# B&R Automation Studio project Parker_BMM_ST_V5_3147_V12 (part 24)

#### calib.c
```c
/********************************************************************
 * COPYRIGHT --  B&R China
 ********************************************************************
 * Program: calib
 * File: calib.c
 * Author: lijianjun
 * Created: March 06, 2013
 ********************************************************************
 * Implementation of program calib --- machine calibn control
 ********************************************************************/

#include <bur/plctypes.h>
#include <string.h>

#ifdef _DEFAULT_INCLUDES
#include <AsDefault.h>
#endif

#include "edge.h"               /*edge function                         */
//#include "keyap880.h"
#include "keyap2100.h"
#include "pic_id.h"
/**************************************************************************************
                            Function Declarations
**************************************************************************************/
void CalibCtrl( Mold_typ *pMold);
void CalibRLCtrl( Mold_typ *pMold);

/**************************************************************************************
**     	        		I N I T U P  O F   T H E   T A S K 		 				     **
**************************************************************************************/
_INIT void calib_init ( void )
{
	t_init = 1;         	/* Disable init step: Don't run init step in first cycle */
	t_stop = 1;				/* Enable stop step:  Run stop step in first cycle */

	Init = 0;
}

/**************************************************************************************
        				C Y C L I C   P A R T   O F   T H E   T A S K
**************************************************************************************/

_CYCLIC void calib_cyclic ( void )
{
	if (0 == t_init)                    /*init step: run only one time after resume  init auto course data  */
	{
		t_init = 1;				        /* Disable init step */
		t_stop = 0;

		gTKcalib.Status = 1;

	}/* if(t_init == 0 ) */

	/*auto solution  */
	gTKcalib.Active++;                  /*  task wait status number */
	/*  ---------------------------------- scan code ------------------------------------------ */
	if(1 == gMachineIn.MainControl && gPanelObj.GetPicture != PIC_INIT && gPanelObj.GetPicture != PIC_SCREEN_SAVE )
	{
		/*  key stop or not  */
		gMachineIn.CalibMode = 1;
		if(PIC_OPTION == gPanelObj.GetPicture)
		{
			if(1 == EDGEPOS(gPanelObj.KeyMatric[S$KEYMATRIX_F12],PKeyMatric[S$KEYMATRIX_F12]))
				{
				RMold.AutoStep			   = 30000;
				RMold.ResetStep			= 30000;
				RMold.LowBlow.Step		= 30000;
				RMold.HighBlow.Step		= 30000;
				RMold.BlowPin.Step		= 30000;
				RMold.BlowPin2.Step		= 30000;
				if(RMold.Carriage.Step < 18000 || RMold.Carriage.Step > 19000)RMold.Carriage.Step = 30000;
				RMold.Clamp.Step		   = 30000;
				//	RMold.CoolPin.Step	   = 30000;
				RMold.CoolPinBlow.Step	= 30000;
				RMold.BlowDeflash.Step	= 30000;
				RMold.Cutter.Step		   = 30000;
				RMold.TopDeflash.Step	= 30000;
				RMold.BottomDeflash.Step= 30000;
				RMold.SupportAir.Step	= 30000;
				RMold.SupportSuckAir.Step	= 30000;
				RMold.ExtrLift.Step		= 30000;
				RMold.Lock.Step			= 30000;
				RMold.PullBottom.Step	= 30000;
				RMold.InnerPin.Step	   = 30000;
				RMold.CutNeck.Step	   = 30000;
				//	RMold.Robot.Step	      = 30000;
				RMold.ChuteDeflashBlow.Step = 30000;
				RMold.SubMold.Step	   = 30000;
				RMold.CoolPin2Blow.Step	= 30000;
				RMold.CoolPin3Blow.Step	= 30000;

				gMacOption.Station  = 0;
			}

			if(1 == EDGEPOS(gPanelObj.KeyMatric[S$KEYMATRIX_F13],PKeyMatric[S$KEYMATRIX_F13]))
				{
				LMold.AutoStep			   = 30000;
				LMold.ResetStep			= 30000;
				LMold.LowBlow.Step		= 30000;
				LMold.HighBlow.Step		= 30000;
				LMold.BlowPin.Step		= 30000;
				LMold.BlowPin2.Step		= 30000;
				LMold.CoolPinBlow.Step	= 30000;
				if(LMold.Carriage.Step < 18000 || LMold.Carriage.Step > 19000)LMold.Carriage.Step	= 30000;
				LMold.Clamp.Step		   = 30000;
				//	LMold.CoolPin.Step	   = 30000;
				LMold.BlowDeflash.Step	= 30000;
				LMold.Cutter.Step		   = 30000;
				LMold.TopDeflash.Step	= 30000;
				LMold.BottomDeflash.Step= 30000;
				LMold.SupportAir.Step	= 30000;
				LMold.SupportSuckAir.Step	= 30000;
				LMold.ExtrLift.Step		= 30000;
				LMold.Lock.Step			= 30000;
				LMold.PullBottom.Step	= 30000;
				LMold.InnerPin.Step	   = 30000;
				LMold.CutNeck.Step	   = 30000;
				//	LMold.Robot.Step	      = 30000;
				LMold.ChuteDeflashBlow.Step = 30000;
				LMold.SubMold.Step	   = 30000;
				LMold.CoolPin2Blow.Step	= 30000;
				LMold.CoolPin3Blow.Step	= 30000;

				gMacOption.Station = 1;
			}

			if(1 == EDGEPOS(gPanelObj.KeyMatric[S$KEYMATRIX_F14],PKeyMatric[S$KEYMATRIX_F14]))
				{
				LMold.AutoStep			   = 30000;
				LMold.ResetStep			= 30000;
				LMold.LowBlow.Step		= 30000;
				LMold.HighBlow.Step	   = 30000;
				LMold.BlowPin.Step		= 30000;
				LMold.BlowPin2.Step		= 30000;
				if(LMold.Carriage.Step < 18000 || LMold.Carriage.Step > 19000)LMold.Carriage.Step	= 30000;
				LMold.Clamp.Step		   = 30000;
				//	LMold.CoolPin.Step	   = 30000;
				LMold.CoolPinBlow.Step	= 30000;
				LMold.BlowDeflash.Step	= 30000;
				LMold.Cutter.Step	      = 30000;
				LMold.TopDeflash.Step	= 30000;
				LMold.BottomDeflash.Step= 30000;
				LMold.SupportAir.Step	= 30000;
				LMold.SupportSuckAir.Step	= 30000;
				LMold.ExtrLift.Step		= 30000;
				LMold.Lock.Step			= 30000;
				LMold.PullBottom.Step	= 30000;
				LMold.InnerPin.Step	   = 30000;
				LMold.CutNeck.Step	   = 30000;
				//	LMold.Robot.Step	      = 30000;
				LMold.ChuteDeflashBlow.Step = 30000;
				LMold.SubMold.Step	   = 30000;
				LMold.CoolPin2Blow.Step	= 30000;
				LMold.CoolPin3Blow.Step	= 30000;

				RMold.AutoStep			   = 30000;
				RMold.ResetStep			= 30000;
				RMold.LowBlow.Step		= 30000;
				RMold.HighBlow.Step		= 30000;
				RMold.BlowPin.Step		= 30000;
				RMold.BlowPin2.Step		= 30000;
				if(RMold.Carriage.Step < 18000 || RMold.Carriage.Step > 19000)RMold.Carriage.Step = 30000;
				RMold.Clamp.Step		   = 30000;
				//	RMold.CoolPin.Step  	   = 30000;
				RMold.CoolPinBlow.Step	= 30000;
				RMold.BlowDeflash.Step	= 30000;
				RMold.Cutter.Step		   = 30000;
				RMold.TopDeflash.Step	= 30000;
				RMold.BottomDeflash.Step= 30000;
				RMold.SupportAir.Step	= 30000;
				RMold.SupportSuckAir.Step	= 30000;
				RMold.ExtrLift.Step		= 30000;
				RMold.Lock.Step			= 30000;
				RMold.PullBottom.Step	= 30000;
				RMold.InnerPin.Step	   = 30000;
				RMold.CutNeck.Step   	= 30000;
				//	RMold.Robot.Step	      = 30000;
				RMold.ChuteDeflashBlow.Step = 30000;
				RMold.SubMold.Step	   = 30000;
				RMold.CoolPin2Blow.Step	= 30000;
				RMold.CoolPin3Blow.Step	= 30000;

				gMacOption.Station  = 2;
			}
		}/* if(PIC_OPTION == gPanelObj.GetPicture) */

		if(1 == gMachineFix.Option.bHideLeftStation)
		{
			gMacOption.Station = 1;
			RightOption = 1;
			LeftOption = 0;
		}

		if(1 == LeftOption && 0 == LeftOptionOld)
		{
			RightOption = 0;
			LeftRight   = 0;

			RMold.AutoStep			   = 30000;
			RMold.ResetStep			= 30000;
			RMold.LowBlow.Step		= 30000;
			RMold.HighBlow.Step		= 30000;
			RMold.BlowPin.Step		= 30000;
			RMold.BlowPin2.Step		= 30000;
			if(RMold.Carriage.Step < 18000 || RMold.Carriage.Step > 19000)RMold.Carriage.Step = 30000;
			RMold.Clamp.Step		   = 30000;
			//	RMold.CoolPin.Step	   = 30000;
			RMold.CoolPinBlow.Step	= 30000;
			RMold.BlowDeflash.Step	= 30000;
			RMold.Cutter.Step	   	= 30000;
			RMold.TopDeflash.Step	= 30000;
			RMold.BottomDeflash.Step= 30000;
			RMold.SupportAir.Step	= 30000;
			RMold.SupportSuckAir.Step	= 30000;
			RMold.ExtrLift.Step		= 30000;
			RMold.Lock.Step			= 30000;
			RMold.PullBottom.Step	= 30000;
			RMold.InnerPin.Step	   = 30000;
			RMold.CutNeck.Step	   = 30000;
			//	RMold.Robot.Step	      = 30000;
			RMold.SubMold.Step	   = 30000;
			RMold.ChuteDeflashBlow.Step = 30000;
			RMold.CoolPin2Blow.Step	= 30000;
			RMold.CoolPin3Blow.Step	= 30000;
			gMacOption.Station = 0;
		}

		LeftOptionOld = LeftOption;

		if(1 == RightOption && 0 == RightOptionOld)
		{
			LeftOption  = 0;
			LeftRight   = 0;

			LMold.AutoStep			   = 30000;
			LMold.ResetStep	      = 30000;
			LMold.LowBlow.Step		= 30000;
			LMold.HighBlow.Step		= 30000;
			LMold.BlowPin.Step		= 30000;
			LMold.BlowPin2.Step		= 30000;
			LMold.CoolPinBlow.Step	= 30000;
			if(LMold.Carriage.Step < 18000 || LMold.Carriage.Step > 19000)LMold.Carriage.Step = 30000;
			LMold.Clamp.Step		   = 30000;
			//	LMold.CoolPin.Step	   = 30000;
			LMold.BlowDeflash.Step	= 30000;
			LMold.Cutter.Step		   = 30000;
			LMold.TopDeflash.Step	= 30000;
			LMold.BottomDeflash.Step= 30000;
			LMold.SupportAir.Step	= 30000;
			LMold.SupportSuckAir.Step	= 30000;
			LMold.ExtrLift.Step		= 30000;
			LMold.Lock.Step			= 30000;
			LMold.PullBottom.Step	= 30000;
			LMold.InnerPin.Step	   = 30000;
			LMold.CutNeck.Step	   = 30000;
			//	LMold.Robot.Step	      = 30000;
			LMold.ChuteDeflashBlow.Step = 30000;
			LMold.SubMold.Step	   = 30000;
			LMold.CoolPin2Blow.Step	= 30000;
			LMold.CoolPin3Blow.Step	= 30000;

			gMacOption.Station  = 1;
		}

		RightOptionOld = RightOption;

		if(1 == LeftRight && 0 == LeftRightOld)
		{
			LeftOption  = 0;
			RightOption = 0;

			LMold.AutoStep			   = 30000;
			LMold.ResetStep		   = 30000;
			LMold.LowBlow.Step		= 30000;
			LMold.HighBlow.Step		= 30000;
			LMold.BlowPin.Step		= 30000;
			LMold.BlowPin2.Step		= 30000;
			if(LMold.Carriage.Step < 18000 || LMold.Carriage.Step > 19000)LMold.Carriage.Step = 30000;
			LMold.Clamp.Step		   = 30000;
			//	LMold.CoolPin.Step	   = 30000;
			LMold.CoolPinBlow.Step	= 30000;
			LMold.BlowDeflash.Step	= 30000;
			LMold.Cutter.Step		   = 30000;
			LMold.TopDeflash.Step	= 30000;
			LMold.BottomDeflash.Step= 30000;
			LMold.SupportAir.Step	= 30000;
			LMold.SupportSuckAir.Step	= 30000;
			LMold.ExtrLift.Step		= 30000;
			LMold.Lock.Step			= 30000;
			LMold.PullBottom.Step	= 30000;
			LMold.InnerPin.Step	   = 30000;
			LMold.CutNeck.Step	   = 30000;
			//	LMold.Robot.Step	      = 30000;
			LMold.ChuteDeflashBlow.Step	      = 30000;
			LMold.SubMold.Step	   = 30000;
			LMold.CoolPin2Blow.Step	= 30000;
			LMold.CoolPin3Blow.Step	= 30000;

			RMold.AutoStep			   = 30000;
			RMold.ResetStep			= 30000;
			RMold.LowBlow.Step		= 30000;
			RMold.HighBlow.Step	   = 30000;
			RMold.BlowPin.Step		= 30000;
			RMold.BlowPin2.Step		= 30000;
			if(RMold.Carriage.Step < 18000 || RMold.Carriage.Step > 19000)RMold.Carriage.Step	= 30000;
			RMold.Clamp.Step		   = 30000;
			//	RMold.CoolPin.Step  	   = 30000;
			RMold.CoolPinBlow.Step	= 30000;
			RMold.BlowDeflash.Step	= 30000;
			RMold.Cutter.Step		   = 30000;
			RMold.TopDeflash.Step	= 30000;
			RMold.BottomDeflash.Step= 30000;
			RMold.SupportAir.Step	= 30000;
			RMold.SupportSuckAir.Step	= 30000;
			RMold.ExtrLift.Step		= 30000;
			RMold.Lock.Step			= 30000;
			RMold.PullBottom.Step	= 30000;
			RMold.InnerPin.Step	   = 30000;
			RMold.CutNeck.Step  	   = 30000;
			//	RMold.Robot.Step	      = 30000;
			RMold.ChuteDeflashBlow.Step = 30000;
			RMold.SubMold.Step	   = 30000;
			RMold.CoolPin2Blow.Step	= 30000;
			RMold.CoolPin3Blow.Step	= 30000;

			gMacOption.Station = 2;
		}

		LeftRightOld = LeftRight;

		if(0 == gMacOption.Station)
		{
			LeftOption = 1;
			RightOption = 0;
			LeftRight = 0;
		}

		if(1 == gMacOption.Station)
		{
			LeftOption  = 0;
			RightOption = 1;
			LeftRight   = 0;
		}

		if(2 == gMacOption.Station)
		{
			LeftOption  = 0;
			RightOption = 0;
			LeftRight   = 1;
		}

		if(1 == gMachineIn.CalibMode && 0 == gMachineIn.SafeCalibPressure)
		{
			/* ---------------- 左右模动作 ---------------- */
			//1 = 正常模式    0 = hold to run
			if((0 == RightOption) && (1 == LeftOption))
			{
				CalibCtrl(&LMold);
			}

			if((1 == RightOption) && (0 == LeftOption))
			{
				CalibCtrl(&RMold);
			}

			if ((0 == RightOption) && (0 == LeftOption))
			{
				CalibRLCtrl(&RMold);
			}

		}/* if(1 == gMachineIn.CalibMode) */
	}/* if(1 == gMachineIn.MainControl && gPanelObj.GetPicture != PIC_INIT && gPanelObj.GetPicture != PIC_SCREEN_SAVE) */
	/*  --------------------------------------------------------------------------------------- */

	if (1 == gTKcalib.Stop)   /* enable stop step */
	{
		t_stop        = 1;
		gTKcalib.Stop = 0;
	}

	/* auto solution end */
	if(1 == t_stop)
	{
		//	memset(&LMold.ValveOut,0,sizeof(LMold.ValveOut));
		//	memset(&RMold.ValveOut,0,sizeof(RMold.ValveOut));

		//		memset(&gMachineOut.LMold,0,sizeof(gMachineOut.LMold));
		//    	memset(&gMachineOut.RMold,0,sizeof(gMachineOut.RMold));

//		memset(&LMold.ValveOut.ClampCls,0,sizeof(LMold.ValveOut)-12);
//		memset(&RMold.ValveOut.ClampCls,0,sizeof(RMold.ValveOut)-12);

		LMold.BottomDeflash.Step = 30000;
		RMold.BottomDeflash.Step = 30000;

		LMold.HighBlow.Step = 30000;
		RMold.HighBlow.Step = 30000;

		LMold.LowBlow.Step = 30000;
		RMold.LowBlow.Step = 30000;

		LMold.BlowPin.Step = 30000;
		RMold.BlowPin.Step = 30000;

		LMold.BlowPin2.Step = 30000;
		RMold.BlowPin2.Step = 30000;

		LMold.Clamp.Step = 30000;
		RMold.Clamp.Step = 30000;

		LMold.Carriage.Step = 30000;
		RMold.Carriage.Step = 30000;

		LMold.TopDeflash.Step = 30000;
		RMold.TopDeflash.Step = 30000;

		LMold.Plate.Step = 30000;/*Albert*/
		RMold.Plate.Step = 30000;/*Albert*/

		LMold.Carriage.v_set = 0;
		RMold.Carriage.v_set = 0;

		LMold.Clamp.v_set = 0;
		RMold.Clamp.v_set = 0;

		LMold.Clamp.p_set = 0;/*Albert*/
		RMold.Clamp.p_set = 0;/*Albert*/

		LMold.BlowPin.v_set = 0;
		RMold.BlowPin.v_set = 0;

		LMold.TopDeflash.p_set = 0;/*Albert*/
		RMold.TopDeflash.p_set = 0;/*Albert*/

		LMold.Plate.p_set = 0;/*Albert*/
		RMold.Plate.p_set = 0;/*Albert*/

		LMold.BottomDeflash.p_set =0;
		RMold.BottomDeflash.p_set =0;

		LMold.SubMold.Step =30000;
		RMold.SubMold.Step =30000;

		LMold.BottomSubMold.Step =30000;
		RMold.BottomSubMold.Step =30000;

		LMold.SubMold.p_set =0;
		RMold.SubMold.p_set =0;

		LMold.BottomSubMold.p_set =0;
		RMold.BottomSubMold.p_set =0;

		LMold.RobotOpnCls.Step = 30000;
		RMold.RobotOpnCls.Step = 30000;

		LMold.Robot.Step = 30000;
		RMold.Robot.Step = 30000;

		t_init         = 0;                 /* next resume ,enable init step */
		gTKcalib.Status = 0;
		ST_tmp_suspend(0);
	} /* if (t_stop==1) */

}

/* ------------------------------------------------------------------*/
void CalibCtrl( Mold_typ *pMold)
{
	if (1==gMacOption.Station) /*Right mold*/
	{
		/* -------------------  Carriage up   ----------------------*/
		if(1 == EDGEPOS(gPanelObj.KeyMatric[S$KEYMATRIX_CARRIAGE_UP ],PKeyMatric[S$KEYMATRIX_CARRIAGE_UP ]))
		{
			if(1 == gMachineOut.OilPump)
			{
				if( 1 == pMold->TransDIn.ClampOpnLimit || (1 == pMold->TransDIn.BlowPinUpLimit && 1 == pMold->TransDIn.BlowPin2UpLimit))
				{
					if(	1 == pMold->TransDIn.TopDeflashBwLimit
						&& 1 == pMold->TransDIn.BottomDeflashBwLimit
						&& 1 == pMold->TransDIn.SubMoldClsLimit && 1 == pMold->TransDIn.BottomSubMoldClsLimit
						&& 1 == pMold->TransDIn.HookPinBwLimit)
					{
						if(((pMold == & LMold) && 1 == RMold.TransDIn.CarriageBwLimit)
							||((pMold == & RMold) && (1 == gMachineFix.Option.bHideLeftStation || 1 == LMold.TransDIn.CarriageBwLimit)))
						{
							pMold->Carriage.Step = 5000;       /* Carriage up calibration */
						}
						else
						{
							if(pMold == & LMold)
							{
								gImply.RCarriageBw = !RMold.TransDIn.CarriageBwLimit;
							}
							else
							{
								gImply.LCarriageBw = !LMold.TransDIn.CarriageBwLimit;
							}
						}
					}
					else
					{
						if(pMold == & LMold)
						{
							gImply.LTopDeflashBw 	= !pMold->TransDIn.TopDeflashBwLimit;
							gImply.LBottomDeflashBw = !pMold->TransDIn.BottomDeflashBwLimit;
							gImply.LSubMoldFw 		= !pMold->TransDIn.SubMoldClsLimit;
							gImply.LBottomSubMoldFw	= !pMold->TransDIn.BottomSubMoldClsLimit;
							gImply.LHookPinBw 		= !pMold->TransDIn.HookPinBwLimit;

						}
						else
						{
							gImply.RTopDeflashBw 	= !pMold->TransDIn.TopDeflashBwLimit;
							gImply.RBottomDeflashBw = !pMold->TransDIn.BottomDeflashBwLimit;
							gImply.RSubMoldFw 		= !pMold->TransDIn.SubMoldClsLimit;
							gImply.RBottomSubMoldFw	= !pMold->TransDIn.BottomSubMoldClsLimit;
							gImply.RHookPinBw 		= !pMold->TransDIn.HookPinBwLimit;
						}
					}
				}
				else
				{
					if(pMold == & LMold)
					{
						gImply.LClampOpn     = !pMold->TransDIn.ClampOpnLimit;
						gImply.LPinUp    	 = !pMold->TransDIn.BlowPinUpLimit;
						gImply.LPin2Up    	 = !pMold->TransDIn.BlowPin2UpLimit;
					}
					else
					{
						gImply.RClampOpn     = !pMold->TransDIn.ClampOpnLimit;
						gImply.RPinUp    	 = !pMold->TransDIn.BlowPinUpLimit;
						gImply.RPin2Up    	 = !pMold->TransDIn.BlowPin2UpLimit;
					}

				}
			}
			else
			{
				gImply.OilPumpNotOn  = !gMachineOut.OilPump;
			}
		}/* if(1 == EDGEPOS(gPanelObj.KeyMatric[S$KEYMATRIX_CARRIAGE_UP  ],PKeyMatric[S$KEYMATRIX_CARRIAGE_UP  ])) */

		if(1 == EDGENEG(gPanelObj.KeyMatric[S$KEYMATRIX_CARRIAGE_UP ],NKeyMatric[S$KEYMATRIX_CARRIAGE_UP]))
		{
			pMold->Carriage.Step = 20000;
		}

		/* -------------------  Carriage down   ----------------------*/
		if(1 == EDGEPOS(gPanelObj.KeyMatric[S$KEYMATRIX_CARRIAGE_DN ],PKeyMatric[S$KEYMATRIX_CARRIAGE_DN ]))
		{
			if(1 == gMachineOut.OilPump)
			{
				if(1 == pMold->TransDIn.BlowPinUpLimit && 1 == pMold->TransDIn.BlowPin2UpLimit)
				{
					if( 1 == pMold->TransDIn.TopDeflashBwLimit
						&& 1 == pMold->TransDIn.BottomDeflashBwLimit
						&& 1 == pMold->TransDIn.CoolPinUpLimit && 1 == pMold->TransDIn.CoolPin2UpLimit && 1==pMold->TransDIn.CoolPin3UpLimit
						&& 1 == pMold->TransDIn.RobotBwLimit
						&& 1 == pMold->TransDIn.ExtRobotUpLmit
						&& 1 == pMold->TransDIn.HookPinBwLimit)
					{
						pMold->Carriage.Step = 15000;       /* Carriage down calibration */
					}
					else
					{
						if(pMold == & LMold)
						{
							gImply.LTopDeflashBw = ! pMold->TransDIn.TopDeflashBwLimit;
							gImply.LBottomDeflashBw = ! pMold->TransDIn.BottomDeflashBwLimit;
							gImply.LCoolPinUp	= !pMold->TransDIn.CoolPinUpLimit;
							gImply.LCoolPin2Up	= !pMold->TransDIn.CoolPin2UpLimit;
							gImply.LCoolPin3Up	= !pMold->TransDIn.CoolPin3UpLimit;
							gImply.LRobotBw		= !pMold->TransDIn.RobotBwLimit;

							gImply.LExtRobotUp 		= !pMold->TransDIn.ExtRobotUpLmit;
							gImply.LHookPinBw 		= !pMold->TransDIn.HookPinBwLimit;
						}
						else
						{
							gImply.RTopDeflashBw = !pMold->TransDIn.TopDeflashBwLimit;
							gImply.RBottomDeflashBw = ! pMold->TransDIn.BottomDeflashBwLimit;
							gImply.RCoolPinUp	= !pMold->TransDIn.CoolPinUpLimit;
							gImply.RCoolPin2Up	= !pMold->TransDIn.CoolPin2UpLimit;
							gImply.RCoolPin3Up	= !pMold->TransDIn.CoolPin3UpLimit;
							gImply.RRobotBw		= !pMold->TransDIn.RobotBwLimit;

							gImply.RExtRobotUp 		= !pMold->TransDIn.ExtRobotUpLmit;
							gImply.RHookPinBw 		= !pMold->TransDIn.HookPinBwLimit;
						}

					}
				}
				else
				{
					if(pMold == & LMold)
					{
						gImply.LPinUp        = !pMold->TransDIn.BlowPinUpLimit;
						gImply.LPin2Up       = !pMold->TransDIn.BlowPin2UpLimit;
					}
					else
					{
						gImply.RPinUp        = !pMold->TransDIn.BlowPinUpLimit;
						gImply.RPin2Up       = !pMold->TransDIn.BlowPin2UpLimit;
					}

				}
			}
			else
			{
				gImply.OilPumpNotOn  = !gMachineOut.OilPump;
			}

		}/* if(1 == EDGEPOS(gPanelObj.KeyMatric[S$KEYMATRIX_CARRIAGE_DN ],PKeyMatric[S$KEYMATRIX_CARRIAGE_DN ]))*/

		if(1 == EDGENEG(gPanelObj.KeyMatric[S$KEYMATRIX_CARRIAGE_DN ],NKeyMatric[S$KEYMATRIX_CARRIAGE_DN ]))
		{
			pMold->Carriage.Step = 20000;
		}
	}
	/*-------------------------------------------------------------------------------------------------------------------*/
	if (0==gMacOption.Station) /*left mold*/
	{
		/* -------------------  Carriage up   ----------------------*/
		if(1 == EDGEPOS(gPanelObj.KeyMatric[S$KEYMATRIX_CARRIAGE_DN ],PKeyMatric[S$KEYMATRIX_CARRIAGE_DN ]))
		{
			if(1 == gMachineOut.OilPump)
			{
				if( 1 == pMold->TransDIn.ClampOpnLimit || (1 == pMold->TransDIn.BlowPinUpLimit && 1 == pMold->TransDIn.BlowPin2UpLimit))
				{
					if(	1 == pMold->TransDIn.TopDeflashBwLimit
						&& 1 == pMold->TransDIn.BottomDeflashBwLimit
						&& 1 == pMold->TransDIn.SubMoldClsLimit && 1 == pMold->TransDIn.BottomSubMoldClsLimit
						&& 1 == pMold->TransDIn.HookPinBwLimit)
					{
						if(((pMold == & LMold) && 1 == RMold.TransDIn.CarriageBwLimit)
							||((pMold == & RMold) && (1 == gMachineFix.Option.bHideLeftStation || 1 == LMold.TransDIn.CarriageBwLimit)))
						{
							pMold->Carriage.Step = 5000;       /* Carriage up calibration */
						}
						else
						{
							if(pMold == & LMold)
							{
								gImply.RCarriageBw = !RMold.TransDIn.CarriageBwLimit;
							}
							else
							{
								gImply.LCarriageBw = !LMold.TransDIn.CarriageBwLimit;
							}
						}
					}
					else
					{
						if(pMold == & LMold)
						{
							gImply.LTopDeflashBw 	= ! pMold->TransDIn.TopDeflashBwLimit;
							gImply.LBottomDeflashBw = !pMold->TransDIn.BottomDeflashBwLimit;
							gImply.LSubMoldFw 		= !pMold->TransDIn.SubMoldClsLimit;
							gImply.LBottomSubMoldFw	= !pMold->TransDIn.BottomSubMoldClsLimit;
							gImply.LHookPinBw 		= !pMold->TransDIn.HookPinBwLimit;
						}
						else
						{
							gImply.RTopDeflashBw 	= ! pMold->TransDIn.TopDeflashBwLimit;
							gImply.RBottomDeflashBw = !pMold->TransDIn.BottomDeflashBwLimit;
							gImply.RSubMoldFw 		= !pMold->TransDIn.SubMoldClsLimit;
							gImply.RBottomSubMoldFw	= !pMold->TransDIn.BottomSubMoldClsLimit;
							gImply.RHookPinBw 		= !pMold->TransDIn.HookPinBwLimit;
						}

					}
				}
				else
				{
					if(pMold == & LMold)
					{
						gImply.LClampOpn     = !pMold->TransDIn.ClampOpnLimit;
						gImply.LPinUp    	 = !pMold->TransDIn.BlowPinUpLimit;
						gImply.LPin2Up    	 = !pMold->TransDIn.BlowPin2UpLimit;
					}
					else
					{
						gImply.RClampOpn     = !pMold->TransDIn.ClampOpnLimit;
						gImply.RPinUp    	 = !pMold->TransDIn.BlowPinUpLimit;
						gImply.RPin2Up    	 = !pMold->TransDIn.BlowPin2UpLimit;
					}

				}
			}
			else
			{
				gImply.OilPumpNotOn  = !gMachineOut.OilPump;
			}
		}/* if(1 == EDGEPOS(gPanelObj.KeyMatric[S$KEYMATRIX_CARRIAGE_DN  ],PKeyMatric[S$KEYMATRIX_CARRIAGE_DN  ])) */

		if(1 == EDGENEG(gPanelObj.KeyMatric[S$KEYMATRIX_CARRIAGE_DN ],NKeyMatric[S$KEYMATRIX_CARRIAGE_DN]))
		{
			pMold->Carriage.Step = 20000;
		}

		/* -------------------  Carriage down   ----------------------*/
		if(1 == EDGEPOS(gPanelObj.KeyMatric[S$KEYMATRIX_CARRIAGE_UP],PKeyMatric[S$KEYMATRIX_CARRIAGE_UP ]))
		{
			if(1 == gMachineOut.OilPump)
			{
				if(1 == pMold->TransDIn.BlowPinUpLimit && 1 == pMold->TransDIn.BlowPin2UpLimit)
				{
					if( 1 == pMold->TransDIn.TopDeflashBwLimit
						&& 1 == pMold->TransDIn.BottomDeflashBwLimit
						&& 1 == pMold->TransDIn.CoolPinUpLimit && 1 == pMold->TransDIn.CoolPin2UpLimit && 1==pMold->TransDIn.CoolPin3UpLimit
						&& 1 == pMold->TransDIn.ExtRobotUpLmit
						&& 1 == pMold->TransDIn.HookPinBwLimit)
					{
						pMold->Carriage.Step = 15000;       /* Carriage down calibration */
					}
					else
					{
						if(pMold == & LMold)
						{
							gImply.LPinUp        = !pMold->TransDIn.BlowPinUpLimit;
							gImply.LTopDeflashBw = ! pMold->TransDIn.TopDeflashBwLimit;
							gImply.LBottomDeflashBw = ! pMold->TransDIn.BottomDeflashBwLimit;
							gImply.LCoolPinUp	= !pMold->TransDIn.CoolPinUpLimit;
							gImply.LCoolPin2Up	= !pMold->TransDIn.CoolPin2UpLimit;
							gImply.LCoolPin3Up	= !pMold->TransDIn.CoolPin3UpLimit;

							gImply.LExtRobotUp 		= !pMold->TransDIn.ExtRobotUpLmit;
							gImply.LHookPinBw 		= !pMold->TransDIn.HookPinBwLimit;

						}
						else
						{
							gImply.RPinUp        = !pMold->TransDIn.BlowPinUpLimit;
							gImply.RTopDeflashBw = !pMold->TransDIn.TopDeflashBwLimit;
							gImply.RBottomDeflashBw = ! pMold->TransDIn.BottomDeflashBwLimit;
							gImply.RCoolPinUp	= !pMold->TransDIn.CoolPinUpLimit;
							gImply.RCoolPin2Up	= !pMold->TransDIn.CoolPin2UpLimit;
							gImply.RCoolPin3Up	= !pMold->TransDIn.CoolPin3UpLimit;

							gImply.RExtRobotUp 		= !pMold->TransDIn.ExtRobotUpLmit;
							gImply.RHookPinBw 		= !pMold->TransDIn.HookPinBwLimit;

						}

					}
				}
				else
				{
					if(pMold == & LMold)
					{
						gImply.LPinUp        = !pMold->TransDIn.BlowPinUpLimit;
						gImply.LPin2Up       = !pMold->TransDIn.BlowPin2UpLimit;
					}
					else
					{
						gImply.RPinUp        = !pMold->TransDIn.BlowPinUpLimit;
						gImply.RPin2Up       = !pMold->TransDIn.BlowPin2UpLimit;
					}

				}
			}
			else
			{
				gImply.OilPumpNotOn  = !gMachineOut.OilPump;
			}

		}/* if(1 == EDGEPOS(gPanelObj.KeyMatric[S$KEYMATRIX_CARRIAGE_UP ],PKeyMatric[S$KEYMATRIX_CARRIAGE_UP ]))*/

		if(1 == EDGENEG(gPanelObj.KeyMatric[S$KEYMATRIX_CARRIAGE_UP ],NKeyMatric[S$KEYMATRIX_CARRIAGE_UP ]))
		{
			pMold->Carriage.Step = 20000;
		}
	}

	/*-------------------------------------------------------------------------------------------------------------------*/

	/* -------------------  open  clamp  ----------------------*/
	if(1 == EDGEPOS(gPanelObj.KeyMatric[S$KEYMATRIX_CLAMP_OPN ],PKeyMatric[S$KEYMATRIX_CLAMP_OPN ]))
	{
		if(1 == gMachineOut.OilPump)
		{
			if( 1 == pMold->TransDIn.TopDeflashBwLimit
				&& 1 == pMold->TransDIn.BottomDeflashBwLimit
				&& 1 == pMold->TransDIn.ExtRobotUpLmit)
			{
				pMold->Clamp.Step = 15000;		/*   clamp open calibration   */
			}
			else
			{
				if(pMold == & LMold)
				{
					gImply.LTopDeflashBw 	= !pMold->TransDIn.TopDeflashBwLimit;
					gImply.LBottomDeflashBw = !pMold->TransDIn.BottomDeflashBwLimit;

					gImply.LExtRobotUp 		= !pMold->TransDIn.ExtRobotUpLmit;
				}
				else
				{
					gImply.RTopDeflashBw 	= ! pMold->TransDIn.TopDeflashBwLimit;
					gImply.RBottomDeflashBw = ! pMold->TransDIn.BottomDeflashBwLimit;

					gImply.RExtRobotUp 		= !pMold->TransDIn.ExtRobotUpLmit;

				}
			}
		}
		else
		{
			gImply.OilPumpNotOn  = !gMachineOut.OilPump;
		}

	}

	if(1 == EDGENEG(gPanelObj.KeyMatric[S$KEYMATRIX_CLAMP_OPN ],NKeyMatric[S$KEYMATRIX_CLAMP_OPN ]))
	{
		if(pMold == & LMold)
		{
			gLClampOpnFlag_Calib =0;
		}
		else
		{
			gRClampOpnFlag_Calib =0;
		}

		pMold->Clamp.Step = 20000;
	}

	/* -------------------  close  clamp  ----------------------*/
	if(1 == EDGEPOS(gPanelObj.KeyMatric[S$KEYMATRIX_CLAMP_CLS ],PKeyMatric[S$KEYMATRIX_CLAMP_CLS ]))
	{
		if(1 == gMachineOut.OilPump)
		{
			if(1 == pMold->TransDIn.CarriageFwLimit || (1 == pMold->TransDIn.BlowPinUpLimit && 1 == pMold->TransDIn.BlowPin2UpLimit))
			{
				if( 1 == pMold->TransDIn.CoolPinUpLimit
					&& 1 == pMold->TransDIn.SubMoldClsLimit
					&& 1 == pMold->TransDIn.BottomSubMoldClsLimit
					&& 1 == pMold->TransDIn.RobotBwLimit)
				{
					pMold->Clamp.Step = 5000;		/*   clamp close calibration   */
				}
				else
				{
					if(pMold == & LMold)
					{
						gImply.LCoolPinUp = !pMold->TransDIn.CoolPinUpLimit;

						gImply.LSubMoldFw 		= !pMold->TransDIn.SubMoldClsLimit;
						gImply.LBottomSubMoldFw	= !pMold->TransDIn.BottomSubMoldClsLimit;
						gImply.LRobotBw		= !pMold->TransDIn.RobotBwLimit;

					}
					else
					{
						gImply.RCoolPinUp = !pMold->TransDIn.CoolPinUpLimit;

						gImply.RSubMoldFw 		= !pMold->TransDIn.SubMoldClsLimit;
						gImply.RBottomSubMoldFw = !pMold->TransDIn.BottomSubMoldClsLimit;
						gImply.RRobotBw		= !pMold->TransDIn.RobotBwLimit;

					}/* if(pMold == & LMold) */
				}
			}
			else
			{
				if(pMold == & LMold)
				{
					gImply.LCarriageFw	 = !pMold->TransDIn.CarriageFwLimit;
					gImply.LPinUp        = !pMold->TransDIn.BlowPinUpLimit;
					gImply.LPin2Up       = !pMold->TransDIn.BlowPin2UpLimit;
				}
				else
				{
					gImply.RCarriageFw	 = !pMold->TransDIn.CarriageFwLimit;
					gImply.RPinUp        = !pMold->TransDIn.BlowPinUpLimit;
					gImply.RPin2Up       = !pMold->TransDIn.BlowPin2UpLimit;
				}
			}
		}
		else
		{
			gImply.OilPumpNotOn  = !gMachineOut.OilPump;
		}
	}

	if(1 == EDGENEG(gPanelObj.KeyMatric[S$KEYMATRIX_CLAMP_CLS ],NKeyMatric[S$KEYMATRIX_CLAMP_CLS ]))
		{
		if(pMold == & LMold)
		{
			gLClampOpnFlag_Calib =0;
		}
		else
		{
			gRClampOpnFlag_Calib =0;
		}
		pMold->Clamp.Step = 20000;
	}

	/* -------------------   blow pin up  ----------------------*/
	if(1 == EDGEPOS(gPanelObj.KeyMatric[S$KEYMATRIX_BLOWPIN_UP ],PKeyMatric[S$KEYMATRIX_BLOWPIN_UP ]))
	{
		if (1 == gMachineOut.OilPump)
		{
			if(pMold->Option.BlowPin)
			{
				pMold->BlowPin.Step = 15000;
			}

			if(pMold->Option.BlowPin2)
			{
				pMold->BlowPin2.Step = 15000;
			}
		}
		else
		{
			gImply.OilPumpNotOn  = !gMachineOut.OilPump;
		}
	}

	if(1 == EDGENEG(gPanelObj.KeyMatric[S$KEYMATRIX_BLOWPIN_UP ],NKeyMatric[S$KEYMATRIX_BLOWPIN_UP ]))
	{
		pMold->BlowPin.Step = 20000;
		pMold->BlowPin2.Step = 20000;
	}
	/* -------------------   blow pin down  ----------------------*/
	if(1 == EDGEPOS(gPanelObj.KeyMatric[S$KEYMATRIX_BLOWPIN_DN ],PKeyMatric[S$KEYMATRIX_BLOWPIN_DN ]))
	{
		if(1 == gMachineOut.OilPump)
		{
			if(( 1 == pMold->TransDIn.CarriageFwLimit || 1 == pMold->TransDIn.CarriageBwLimit) )
			{
				if(1 == pMold->TransDIn.SubMoldClsLimit
					&& 1 == pMold->TransDIn.BottomSubMoldClsLimit )
				{
					if(pMold->Option.BlowPin)
					{
						pMold->BlowPin.Step = 5000;	/*  blow pin down  */
					}

					if(pMold->Option.BlowPin2)
					{
						pMold->BlowPin2.Step = 5000; /*  blow pin down  */
					}
				}
				else
				{
					if(pMold == & LMold)
					{
						gImply.LSubMoldFw 		= !pMold->TransDIn.SubMoldClsLimit;
						gImply.LBottomSubMoldFw = !pMold->TransDIn.BottomSubMoldClsLimit;

					}
					else
					{
						gImply.RSubMoldFw 		= !pMold->TransDIn.SubMoldClsLimit;
						gImply.RBottomSubMoldFw = !pMold->TransDIn.BottomSubMoldClsLimit;

					}
				}
			}
			else
			{
				if(pMold == & LMold)
				{
					gImply.LCarriageFwBw = !(pMold->TransDIn.CarriageBwLimit || pMold->TransDIn.CarriageFwLimit);
				}
				else
				{
					gImply.RCarriageFwBw = !(pMold->TransDIn.CarriageBwLimit || pMold->TransDIn.CarriageFwLimit);
				}
			}
		}
		else
		{
			gImply.OilPumpNotOn  = !gMachineOut.OilPump;
		}
	}
	if(1 == EDGENEG(gPanelObj.KeyMatric[S$KEYMATRIX_BLOWPIN_DN   ],NKeyMatric[S$KEYMATRIX_BLOWPIN_DN ]))
	{
		pMold->BlowPin.Step = 20000;
		pMold->BlowPin2.Step = 20000;
	}

	/* ------------------------------  pin part forward ----------------------------- */
	if(1 == EDGEPOS(gPanelObj.KeyMatric[S$KEYMATRIX_PIN_PART_FW ],PKeyMatric[S$KEYMATRIX_PIN_PART_FW ]))
		{
		if(pMold->Option.PinPart)
		{
			if(1 == pMold->TransDIn.BlowPinUpLimit)
			{
				pMold->PinPart.Step = 300;
			}
			else
			{
				if(pMold == & LMold)
				{
					gImply.LPinUp = !pMold->TransDIn.BlowPinUpLimit;
				}
				else
				{
					gImply.RPinUp = !pMold->TransDIn.BlowPinUpLimit;
				}
			}
		}
	}

	if(1 == EDGENEG(gPanelObj.KeyMatric[S$KEYMATRIX_PIN_PART_FW ],NKeyMatric[S$KEYMATRIX_PIN_PART_FW ]))
		{
		pMold->PinPart.Step = 20000;
	}

	/* ------------------------------  pin part backward ----------------------------- */
	if(1 == EDGEPOS(gPanelObj.KeyMatric[S$KEYMATRIX_PIN_PART_BW   ],PKeyMatric[S$KEYMATRIX_PIN_PART_BW   ]))
	{
		if(pMold->Option.PinPart)
		{
			if(1 == pMold->TransDIn.BlowPinUpLimit)
			{
				pMold->PinPart.Step = 10300;
			}
			else
			{
				if(pMold == & LMold)
				{
					gImply.LPinUp = !pMold->TransDIn.BlowPinUpLimit;
				}
				else
				{
					gImply.RPinUp = !pMold->TransDIn.BlowPinUpLimit;
				}
			}
		}
	}

	if(1 == EDGENEG(gPanelObj.KeyMatric[S$KEYMATRIX_PIN_PART_BW   ],NKeyMatric[S$KEYMATRIX_PIN_PART_BW   ]))
	{
		pMold->PinPart.Step = 20000;
	}

	/* ------------------------------  Sub mold open ----------------------------- */
	if(1 == EDGEPOS(gPanelObj.KeyMatric[S$KEYMATRIX_SUBMOLD_OPN   ],PKeyMatric[S$KEYMATRIX_SUBMOLD_OPN   ]))
	{
		if(1 == pMold->Option.SubMold )
		{
			if(1 == gMachineOut.OilPump)
			{
				if (1==pMold->Clamp.OpnOverHalf && 1 == pMold->TransDIn.CarriageBwLimit) // 大於微開模
				{
					pMold->SubMold.Step = 15000;
				}
				else
				{
					if(pMold == & LMold)
					{
						gImply.L_SubmoldOut_Clamp = !pMold->Clamp.OpnOverHalf;
						gImply.LCarriageBw = !pMold->TransDIn.CarriageBwLimit;
					}
					else
					{
						gImply.R_SubmoldOut_Clamp = !pMold->Clamp.OpnOverHalf;
						gImply.RCarriageBw = !pMold->TransDIn.CarriageBwLimit;
					}
				}

			}
			else
			{
				gImply.OilPumpNotOn  = !gMachineOut.OilPump;
			}
		}
		else
		{
			gImply.NoFunction = 1;
		}
	}

	if(1 == EDGENEG(gPanelObj.KeyMatric[S$KEYMATRIX_SUBMOLD_OPN   ],NKeyMatric[S$KEYMATRIX_SUBMOLD_OPN   ]))
	{
		pMold->SubMold.Step = 20000;
	}

	/* ------------------------------  sub mold close ----------------------------- */
	if(1 == EDGEPOS(gPanelObj.KeyMatric[S$KEYMATRIX_SUBMOLD_CLS   ],PKeyMatric[S$KEYMATRIX_SUBMOLD_CLS   ]))
	{
		if(pMold->Option.SubMold)
		{
			if(1 == gMachineOut.OilPump)
			{
				pMold->SubMold.Step = 5000;
			}
			else
			{
				gImply.OilPumpNotOn  = !gMachineOut.OilPump;
			}
		}
		else
		{
			gImply.NoFunction = 1;
		}
	}

	if(1 == EDGENEG(gPanelObj.KeyMatric[S$KEYMATRIX_SUBMOLD_CLS   ],NKeyMatric[S$KEYMATRIX_SUBMOLD_CLS   ]))
	{
		pMold->SubMold.Step = 20000;
	}

	/* ------------------------------  Bottom Sub mold open ----------------------------- */
	if(1 == EDGEPOS(gPanelObj.KeyMatric[S$KEYMATRIX_BOTSUBMOLD_OPN  ],PKeyMatric[S$KEYMATRIX_BOTSUBMOLD_OPN  ]))
	{
		if(pMold->Option.BottomSubMold)
		{
			if(1 == gMachineOut.OilPump)
			{
				if (1 == pMold->Clamp.OpnOverHalf && 1 == pMold->TransDIn.CarriageBwLimit)
				{
					pMold->BottomSubMold.Step = 15000;
				}
				else
				{
					if(pMold == & LMold)
					{
						gImply.L_SubmoldOut_Clamp = !pMold->Clamp.OpnOverHalf;
						gImply.LCarriageBw = !pMold->TransDIn.CarriageBwLimit;
					}
					else
					{
						gImply.R_SubmoldOut_Clamp = !pMold->Clamp.OpnOverHalf;
						gImply.RCarriageBw = !pMold->TransDIn.CarriageBwLimit;
					}
				}
			}
			else
			{
				gImply.OilPumpNotOn  = !gMachineOut.OilPump;
			}
		}
		else
		{
			gImply.NoFunction = 1;
		}
	}

	if(1 == EDGENEG(gPanelObj.KeyMatric[S$KEYMATRIX_BOTSUBMOLD_OPN  ],NKeyMatric[S$KEYMATRIX_BOTSUBMOLD_OPN  ]))
	{
		pMold->BottomSubMold.Step = 20000;
	}

	/* ------------------------------ Bottom sub mold close ----------------------------- */
	if(1 == EDGEPOS(gPanelObj.KeyMatric[S$KEYMATRIX_BOTSUBMOLD_CLS  ],PKeyMatric[S$KEYMATRIX_BOTSUBMOLD_CLS  ]))
	{
		if(pMold->Option.BottomSubMold)
		{
			if(1 == gMachineOut.OilPump)
			{
				pMold->BottomSubMold.Step = 5000;
			}
			else
			{
				gImply.OilPumpNotOn  = !gMachineOut.OilPump;
			}
		}
		else
		{
			gImply.NoFunction = 1;
		}
	}
	if(1 == EDGENEG(gPanelObj.KeyMatric[S$KEYMATRIX_BOTSUBMOLD_CLS  ],NKeyMatric[S$KEYMATRIX_BOTSUBMOLD_CLS  ]))
	{
		pMold->BottomSubMold.Step = 20000;
	}

	/* ------------------------------  Screw forward ----------------------------- */
	if(1 == EDGEPOS(gPanelObj.KeyMatric[S$KEYMATRIX_SCREW_FW   ],PKeyMatric[S$KEYMATRIX_SCREW_FW   ]))
	{
		pMold->Screw.Step = 300;
	}

	if(1 == EDGENEG(gPanelObj.KeyMatric[S$KEYMATRIX_SCREW_FW   ],NKeyMatric[S$KEYMATRIX_SCREW_FW   ]))
	{
		pMold->Screw.Step = 20000;
	}

	/* ------------------------------  screw backward ----------------------------- */
	if(1 == EDGEPOS(gPanelObj.KeyMatric[S$KEYMATRIX_SCREW_BW   ],PKeyMatric[S$KEYMATRIX_SCREW_BW   ]))
	{
		pMold->Screw.Step = 10300;
	}

	if(1 == EDGENEG(gPanelObj.KeyMatric[S$KEYMATRIX_SCREW_BW   ],NKeyMatric[S$KEYMATRIX_SCREW_BW   ]))
	{
		pMold->Screw.Step = 20000;
	}

	/* ------------------------------  Top Deflasher forward ----------------------------- */
	if(1 == EDGEPOS(gPanelObj.KeyMatric[S$KEYMATRIX_TOP_DEFLASH_FW  ],PKeyMatric[S$KEYMATRIX_TOP_DEFLASH_FW  ]))
	{
		if(pMold->Option.TopDeflash)
		{
			if(1 == gMachineOut.OilPump)
			{
				if(1 == pMold->TransDIn.CarriageBwLimit
					&& 1 == pMold->Clamp.ClsPos
					&& 1 == pMold->TransDIn.TopDeflashOpnLimit
					&& 1 == pMold->TransDIn.CoolPinUpLimit)
				{
					pMold->TopDeflash.Step = 5000;
				}
				else
				{
					if(pMold == & LMold)
					{
						gImply.LCarriageBw	= !pMold->TransDIn.CarriageBwLimit;
						gImply.LClampCls	= !pMold->Clamp.ClsPos;
						gImply.LTopDeflashOpn	= !pMold->TransDIn.TopDeflashOpnLimit;
						gImply.LCoolPinUp	= !pMold->TransDIn.CoolPinUpLimit;
					}
					else
					{
						gImply.RCarriageBw	= !pMold->TransDIn.CarriageBwLimit;
						gImply.RClampCls	= !pMold->Clamp.ClsPos;
						gImply.RTopDeflashOpn	= !pMold->TransDIn.TopDeflashOpnLimit;
						gImply.RCoolPinUp	= !pMold->TransDIn.CoolPinUpLimit;
					}
				}
			}
			else
			{
				gImply.OilPumpNotOn  = !gMachineOut.OilPump;
			}
		}
		else
		{
			gImply.NoFunction = 1;
		}

	}

	if( ACTUATOR_HYD  == gMachineFix.MoldR.TopDeflash.eActuatorType )
	{
		if(1 == EDGENEG(gPanelObj.KeyMatric[S$KEYMATRIX_TOP_DEFLASH_FW],NKeyMatric[S$KEYMATRIX_TOP_DEFLASH_FW]))
			{
			pMold->TopDeflash.Step = 20000;
		}
	}

	/* ------------------------------ Top Deflasher backward ----------------------------- */
	if(1 == EDGEPOS(gPanelObj.KeyMatric[S$KEYMATRIX_TOP_DEFLASH_BW  ],PKeyMatric[S$KEYMATRIX_TOP_DEFLASH_BW  ]))
	{
		if(pMold->Option.TopDeflash)
		{
			if(1 == gMachineOut.OilPump)
			{
				if(1 == pMold->TransDIn.TopDeflashOpnLimit)
				{
					pMold->TopDeflash.Step = 15000;
				}
				else
				{
					if(pMold == & LMold)
					{
						gImply.LTopDeflashOpn	= !pMold->TransDIn.TopDeflashOpnLimit;
					}
					else
					{
						gImply.RTopDeflashOpn	= !pMold->TransDIn.TopDeflashOpnLimit;
					}
				}
			}
			else
			{
				gImply.OilPumpNotOn  = !gMachineOut.OilPump;
			}
		}
		else
		{
			gImply.NoFunction = 1;
		}
	}

	if( ACTUATOR_HYD  == gMachineFix.MoldR.TopDeflash.eActuatorType )
	{
		if(1 == EDGENEG(gPanelObj.KeyMatric[S$KEYMATRIX_TOP_DEFLASH_BW],NKeyMatric[S$KEYMATRIX_TOP_DEFLASH_BW]))
			{
			pMold->TopDeflash.Step = 20000;
		}
	}

	/* ------------------------------  Bottom Deflasher Forward ----------------------------- */
	if(1 == EDGEPOS(gPanelObj.KeyMatric[S$KEYMATRIX_BOT_DEFLASH_FW],PKeyMatric[S$KEYMATRIX_BOT_DEFLASH_FW]))
	{
		if(pMold->Option.BottomDeflash)
		{
			if(1 == gMachineOut.OilPump)
			{
				if(1 == pMold->TransDIn.CarriageBwLimit && 1 == pMold->Clamp.ClsPos)
				{
					pMold->BottomDeflash.Step = 5000;
				}
				else
				{
					if(pMold == & LMold)
					{
						gImply.LCarriageBw	= !pMold->TransDIn.CarriageBwLimit;
						gImply.LClampCls	= !pMold->Clamp.ClsPos;
					}
					else
					{
						gImply.RCarriageBw	= !pMold->TransDIn.CarriageBwLimit;
						gImply.RClampCls	= !pMold->Clamp.ClsPos;
					}
				}
			}
			else
			{
				gImply.OilPumpNotOn  = !gMachineOut.OilPump;
			}
		}
		else
		{
			gImply.NoFunction = 1;
		}

	}

	if(1 == EDGENEG(gPanelObj.KeyMatric[S$KEYMATRIX_BOT_DEFLASH_FW],NKeyMatric[S$KEYMATRIX_BOT_DEFLASH_FW]))
	{
		pMold->BottomDeflash.Step = 20000;
	}

	/* ------------------------------  Bottom Deflasher Backward ----------------------------- */
	if(1 == EDGEPOS(gPanelObj.KeyMatric[S$KEYMATRIX_BOT_DEFLASH_BW],PKeyMatric[S$KEYMATRIX_BOT_DEFLASH_BW]))
	{
		if(pMold->Option.BottomDeflash)
		{
			if(1 == gMachineOut.OilPump)
			{
				pMold->BottomDeflash.Step = 15000;
			}
			else
			{
				gImply.OilPumpNotOn  = !gMachineOut.OilPump;
			}
		}
		else
		{
			gImply.NoFunction = 1;
		}

	}

	if(1 == EDGENEG(gPanelObj.KeyMatric[S$KEYMATRIX_BOT_DEFLASH_BW],NKeyMatric[S$KEYMATRIX_BOT_DEFLASH_BW]))
	{
		pMold->BottomDeflash.Step = 20000;
	}

	/* ------------------------------  Pull Bottom Forward ----------------------------- */
	if(1 == EDGEPOS(gPanelObj.KeyMatric[S$KEYMATRIX_PULL_BOTTOM_FW],PKeyMatric[S$KEYMATRIX_PULL_BOTTOM_FW]))
		{
		if(pMold->Option.PullBottom)
		{
			if(1 == gMachineOut.OilPump)
			{
				if( 5000 == pMold->PullBottom.Step )
				{
					pMold->PullBottom.Step = 20000;
				}
				else
				{
					pMold->PullBottom.Step = 5000;
				}
			}
			else
			{
				gImply.OilPumpNotOn  = !gMachineOut.OilPump;
			}
		}
		else
		{
			gImply.NoFunction = 1;
		}

	}

	//	if(1 == EDGENEG(gPanelObj.KeyMatric[S$KEYMATRIX_PULL_BOTTOM_FW],NKeyMatric[S$KEYMATRIX_PULL_BOTTOM_FW]))
	//	{
	//		pMold->PullBottom.Step = 20000;
	//	}

	/* ------------------------------  Pull Bottom Backward ----------------------------- */
	//	if(1 == EDGEPOS(gPanelObj.KeyMatric[S$KEYMATRIX_PULL_BOTTOM_BW],PKeyMatric[S$KEYMATRIX_PULL_BOTTOM_BW]))
	//	{
	//		if(pMold->Option.PullBottom)
	//		{
	//			if(1 == gMachineOut.OilPump)
	//			{
	//				pMold->PullBottom.Step = 15000;
	//			}
	//			else
	//			{
	//				gImply.OilPumpNotOn  = !gMachineOut.OilPump;
	//			}
	//		}
	//		else
	//		{
	//			gImply.NoFunction = 1;
	//		}
	//	}
	//
	//	if(1 == EDGENEG(gPanelObj.KeyMatric[S$KEYMATRIX_PULL_BOTTOM_BW],NKeyMatric[S$KEYMATRIX_PULL_BOTTOM_BW]))
	//	{
	//		pMold->PullBottom.Step = 20000;
	//	}

	/* ------------------------------  cutter neck ----------------------------- */
	if(1 == EDGEPOS(gPanelObj.KeyMatric[S$KEYMATRIX_CUT_NECK],PKeyMatric[S$KEYMATRIX_CUT_NECK]))
		{
		if(1 == gMachineIn.SafeGate)
		{
			if(pMold->Option.CutNeck)
			{
				pMold->ValveOut.CutNeck = !pMold->ValveOut.CutNeck;
				pMold->ActInfo.CutNeck  = pMold->ValveOut.CutNeck;
			}
			else
			{
				gImply.NoFunction = 1;
			}
		}
		else
		{
			gImply.SafeGate = 1;
		}
	}

	/*  ------------------------ Robot-Transfer ActuatorType -----------------------  */
	if( ACTUATOR_PNEU  == gMachineFix.MoldR.RobotTransfer.eActuatorType ) //Pneu
	{
		/*  ------------------------ Robot-Transfer Forward/Backward - Pneu -----------------------  */
		if(1 == EDGEPOS(gPanelObj.KeyMatric[S$KEYMATRIX_ROBOT_FW ],PKeyMatric[S$KEYMATRIX_ROBOT_FW ]))
			{
			if(pMold->Option.RobotTransfer)
			{
				if( 1 == gMachineIn.SafeGate && 1 == gMachineOut.OilPump )
				{
					if(0 == pMold->ValveOut.RobotFw)  // Fw
					{
						if( /*1 == pMold->Carriage.BwPos*/
							/*&&*/ 1 == pMold->TransDIn.TopDeflashBwLimit
							&& 1 == pMold->TransDIn.BottomDeflashBwLimit
							&& 1 == pMold->TransDIn.RobotOpnLimit)
						{
							pMold->Robot.Step = 5000;
						}
						else
						{
							if(pMold == & LMold)
							{
								//								gImply.LCarriageBw		= !pMold->Carriage.BwPos;
								gImply.LTopDeflashBw 	= !pMold->TransDIn.TopDeflashBwLimit;
								gImply.LBottomDeflashBw = !pMold->TransDIn.BottomDeflashBwLimit;
								gImply.LRobotOpn 		= !pMold->TransDIn.RobotOpnLimit;
							}
							else
							{
								//								gImply.RCarriageBw		= !pMold->Carriage.BwPos;
								gImply.RTopDeflashBw 	= !pMold->TransDIn.TopDeflashBwLimit;
								gImply.RBottomDeflashBw = !pMold->TransDIn.BottomDeflashBwLimit;
								gImply.RRobotOpn 		= !pMold->TransDIn.RobotOpnLimit;
							}
						}
					}
					else //Bw
					{
						if( 1 == pMold->TransDIn.ClampOpnLimit
							&& 1 == pMold->TransDIn.CoolPin2UpLimit && 1==pMold->TransDIn.CoolPin3UpLimit
							&& 1 == pMold->TransDIn.RobotFwLimit)
						{
							pMold->Robot.Step = 15000;
						}
						else
						{
							if(pMold == & LMold)
							{
								gImply.LClampOpn 	= !pMold->TransDIn.ClampOpnLimit;
								gImply.LCoolPin2Up	= !pMold->TransDIn.CoolPin2UpLimit;
								gImply.LCoolPin3Up	= !pMold->TransDIn.CoolPin3UpLimit;
							}
							else
							{
								gImply.RClampOpn 	= !pMold->TransDIn.ClampOpnLimit;
								gImply.RCoolPin2Up	= !pMold->TransDIn.CoolPin2UpLimit;
								gImply.RCoolPin3Up	= !pMold->TransDIn.CoolPin3UpLimit;
							}
						}
					}
				}
				else
				{
					gImply.OilPumpNotOn  = !gMachineOut.OilPump;
					gImply.SafeGate = !gMachineIn.SafeGate;
				}
			}
			else
			{
				gImply.NoFunction = 1;
			}

		}
	}
	else
	{
		/*  ------------------------Robot-Transfer Forward - Elec/Hyd -----------------------  */
		if(1 == EDGEPOS(gPanelObj.KeyMatric[S$KEYMATRIX_ROBOT_FW ],PKeyMatric[S$KEYMATRIX_ROBOT_FW ]))
			{
			if(pMold->Option.RobotTransfer)
			{
				if(1 == gMachineOut.OilPump)
				{
					//					if(1 == pMold->TransDIn.CarriageBwLimit)
					//					{
					if( 1 == pMold->TransDIn.TopDeflashBwLimit
						&& 1 == pMold->TransDIn.BottomDeflashBwLimit
						&& 1 == pMold->TransDIn.RobotOpnLimit)
					{
						pMold->Robot.Step = 5000;
					}
					else
					{
						if(pMold == & LMold)
						{
							gImply.LTopDeflashBw 	= !pMold->TransDIn.TopDeflashBwLimit;
							gImply.LBottomDeflashBw = !pMold->TransDIn.BottomDeflashBwLimit;
							gImply.LRobotOpn 		= !pMold->TransDIn.RobotOpnLimit;

						}
						else
						{
							gImply.RTopDeflashBw 	= !pMold->TransDIn.TopDeflashBwLimit;
							gImply.RBottomDeflashBw = !pMold->TransDIn.BottomDeflashBwLimit;
							gImply.RRobotOpn 		= !pMold->TransDIn.RobotOpnLimit;

						}
					}
					//					}
					//					else
					//					{
					//						if(pMold == & LMold)
					//						{
					//							gImply.LCarriageBw		= !pMold->TransDIn.CarriageBwLimit;
					//						}
					//						else
					//						{
					//							gImply.RCarriageBw		= !pMold->TransDIn.CarriageBwLimit;
					//						}
					//					}
				}
				else
				{
					gImply.OilPumpNotOn  = !gMachineOut.OilPump;
				}
			}
			else
			{
				gImply.NoFunction = 1;
			}

		}
		if( ACTUATOR_HYD  == gMachineFix.MoldR.RobotTransfer.eActuatorType || ACTUATOR_ELECTRIC  == gMachineFix.MoldR.RobotTransfer.eActuatorType )
		{
			if(1 == EDGENEG(gPanelObj.KeyMatric[S$KEYMATRIX_ROBOT_FW],NKeyMatric[S$KEYMATRIX_ROBOT_FW]))
				{
				pMold->Robot.Step = 20000;
			}
		}
		/*  ------------------------ Robot-Transfer Backward - Elec/Hyd  -----------------------  */
		if(1 == EDGEPOS(gPanelObj.KeyMatric[S$KEYMATRIX_ROBOT_BW],PKeyMatric[S$KEYMATRIX_ROBOT_BW]))
			{
			if(pMold->Option.RobotTransfer)
			{
				if(1 == gMachineOut.OilPump)
				{
					if(1 == pMold->TransDIn.ClampOpnLimit)
					{
						if( 1 == pMold->TransDIn.CoolPin2UpLimit && 1==pMold->TransDIn.CoolPin3UpLimit  )
						{
							pMold->Robot.Step = 15000;

						}
						else
						{
							if(pMold == & LMold)
							{
								gImply.LCoolPin2Up	= !pMold->TransDIn.CoolPin2UpLimit;
								gImply.LCoolPin3Up	= !pMold->TransDIn.CoolPin3UpLimit;

							}
							else
							{
								gImply.RCoolPin2Up	= !pMold->TransDIn.CoolPin2UpLimit;
								gImply.RCoolPin3Up	= !pMold->TransDIn.CoolPin3UpLimit;

							}
						}
					}
					else
					{
						if(pMold == & LMold)
						{
							gImply.LClampOpn = !pMold->Clamp.OpnPos;
						}
						else
						{
							gImply.RClampOpn = !pMold->Clamp.OpnPos;
						}
					}
				}
				else
				{
					gImply.OilPumpNotOn  = !gMachineOut.OilPump;
				}
			}
			else
			{
				gImply.NoFunction = 1;
			}
		}

		if(1 == EDGENEG(gPanelObj.KeyMatric[S$KEYMATRIX_ROBOT_BW],NKeyMatric[S$KEYMATRIX_ROBOT_BW]))
			{
			pMold->Robot.Step = 20000;
		}
	}

	//	/*  ------------------------ robot up -----------------------  */
	//	if(1 == EDGEPOS(gPanelObj.KeyMatric[S$KEYMATRIX_ROBOT_UP],PKeyMatric[S$KEYMATRIX_ROBOT_UP]))
	//	{
	//		if(pMold->Option.RobotUpDn)
	//		{
	//			if(1 == gMachineFix.MoldR.RobotUpDn.eActuatorTyp)
	//			{
	//				pMold->Robot.Step = 15500;
	//			}
	//			else
	//			{
	//				pMold->ActInfo.RobotUp   = 0;
	//				pMold->ValveOut.RobotUp  = 0;
	//
	//				pMold->ActInfo.RobotDn   = 1;
	//				pMold->ValveOut.RobotDn  = 1;
	//			}
	//		}
	//		else
	//		{
	//			gImply.NoFunction = 1;
	//		}
	//	}
	//
	//	if(1 == EDGENEG(gPanelObj.KeyMatric[S$KEYMATRIX_ROBOT_UP],NKeyMatric[S$KEYMATRIX_ROBOT_UP]))
	//	{
	//		if(1 == gMachineFix.MoldR.RobotUpDn.eActuatorTyp)
	//		{
	//			pMold->Robot.Step = 20000;
	//		}
	//		else
	//		{
	//			pMold->ValveOut.RobotFw = 0;
	//			pMold->ActInfo.RobotFw  = 0;
	//
	//			pMold->ValveOut.RobotBw = 0;
	//			pMold->ActInfo.RobotBw  = 0;
	//		}
	//	}
	//
	//
	//	/*  ------------------------ robot down -----------------------  */
	//	if(1 == EDGEPOS(gPanelObj.KeyMatric[S$KEYMATRIX_ROBOT_DN],PKeyMatric[S$KEYMATRIX_ROBOT_DN]))
	//	{
	//		if(pMold->Option.RobotUpDn)
	//		{
	//			if(1 == pMold->TransDIn.RobotBwLimit)
	//			{
	//				if(1 == gMachineFix.MoldR.RobotUpDn.eActuatorTyp)
	//				{
	//					pMold->Robot.Step = 5500;
	//				}
	//				else
	//				{
	//					pMold->ValveOut.RobotDn = !pMold->ValveOut.RobotDn;
	//				}
	//			}
	//			else if(1 == pMold->TransDIn.RobotFwLimit)
	//			{
	//				if(1 == pMold->TransDIn.TopDeflashBwLimit)
	//				{
	//					if(pMold->TransDIn.ClampOpnLimit || pMold->TransDIn.CarriageFwLimit || pMold->TransDIn.CarriageBwLimit)
	//					{
	//						if(1 == gMachineFix.MoldR.RobotUpDn.eActuatorTyp)
	//						{
	//							pMold->Robot.Step = 5500;
	//						}
	//						else
	//						{
	//							pMold->ValveOut.RobotDn = !pMold->ValveOut.RobotDn;
	//						}
	//					}
	//					else
	//					{
	//						if(pMold == & LMold)
	//						{
	//							gImply.LClampOpn   = !pMold->TransDIn.ClampOpnLimit;
	//							gImply.LCarriageBw = !pMold->TransDIn.CarriageBwLimit;
	//							gImply.LCarriageFw = !pMold->TransDIn.CarriageFwLimit;
	//
	//						}
	//						else
	//						{
	//							gImply.RClampOpn   = !pMold->TransDIn.ClampOpnLimit;
	//							gImply.RCarriageBw = !pMold->TransDIn.CarriageBwLimit;
	//							gImply.RCarriageFw = !pMold->TransDIn.CarriageFwLimit;
	//						}
	//					}
	//				}
	//				else
	//				{
	//					if(pMold == & LMold)
	//					{
	//						gImply.LTopDeflashBw = !pMold->TransDIn.TopDeflashBwLimit;
	//					}
	//					else
	//					{
	//						gImply.RTopDeflashBw = !pMold->TransDIn.TopDeflashBwLimit;
	//					}
	//				}
	//			}
	//			else
	//			{
	//				gImply.RRobotFwOrBw = 1;
	//			}
	//		}
	//		else
	//		{
	//			gImply.NoFunction = 1;
	//		}
	//	}
	//
	//	if(1 == EDGENEG(gPanelObj.KeyMatric[S$KEYMATRIX_ROBOT_DN],NKeyMatric[S$KEYMATRIX_ROBOT_DN]))
	//	{
	//		if(1 == gMachineFix.MoldR.RobotUpDn.eActuatorTyp)
	//		{
	//			pMold->Robot.Step = 20000;
	//		}
	//		else
	//		{
	//			pMold->ValveOut.RobotFw = 0;
	//			pMold->ActInfo.RobotFw  = 0;
	//
	//			pMold->ValveOut.RobotBw = 0;
	//			pMold->ActInfo.RobotBw  = 0;
	//		}
	//	}

	/*  ------------------------ Robot Open/Close  -----------------------  */
	if( ACTUATOR_PNEU  == gMachineFix.MoldR.RobotOpnCls.eActuatorType ) //Pneu
	{
		/*  ------------------------ Robot Open/Close - Pneu -----------------------  */
		if(1 == EDGEPOS(gPanelObj.KeyMatric[S$KEYMATRIX_ROBOT_CLS],PKeyMatric[S$KEYMATRIX_ROBOT_CLS]))
			{
			if(pMold->Option.RobotOpnCls)
			{
				if( 1 == gMachineOut.OilPump )
				{
					if(0 == pMold->ValveOut.RobotCls)  //Opn
					{
						if(  1 == pMold->TransDIn.RobotFwLimit || 1 == pMold->TransDIn.RobotBwLimit)
						{
							pMold->RobotOpnCls.Step = 5000;
						}
						else
						{
							if(pMold == & LMold)
							{
								gImply.LRobotFw = !pMold->TransDIn.RobotFwLimit;
								gImply.LRobotBw = !pMold->TransDIn.RobotBwLimit;
							}
							else
							{
								gImply.RRobotFw = !pMold->TransDIn.RobotFwLimit;
								gImply.RRobotBw = !pMold->TransDIn.RobotBwLimit;
							}
						}
					}
					else //Cls
					{
						if(  1 == pMold->TransDIn.RobotFwLimit || 1 == pMold->TransDIn.RobotBwLimit)
						{
							pMold->RobotOpnCls.Step = 15000;
						}
						else
						{
							if(pMold == & LMold)
							{
								gImply.LRobotFw = !pMold->TransDIn.RobotFwLimit;
								gImply.LRobotBw = !pMold->TransDIn.RobotBwLimit;
							}
							else
							{
								gImply.RRobotFw = !pMold->TransDIn.RobotFwLimit;
								gImply.RRobotBw = !pMold->TransDIn.RobotBwLimit;
							}
						}
					}
				}
				else
				{
					gImply.OilPumpNotOn  = !gMachineOut.OilPump;
				}
			}
			else
			{
				gImply.NoFunction = 1;
			}

		}
	}

	/*  ------------------------ Product Aux close -----------------------  */
	//	if(1 == EDGEPOS(gPanelObj.KeyMatric[S$KEYMATRIX_PRODUCTAUX_CLS  ],PKeyMatric[S$KEYMATRIX_PRODUCTAUX_CLS  ]))
	//		{
	//		if (1==gUserPara.bProductAuxClamp)
	//		{
	//			pMold->ValveOut.ProductAuxClamp = !pMold->ValveOut.ProductAuxClamp;
	//			//	pMold->ActInfo.RobotCls  = pMold->ValveOut.ProductAuxClamp;
	//		}
	//		else
	//		{
	//			gImply.NoFunction = 1;
	//		}
	//
	//	}
	/*  ------------------------ sensor up -----------------------  */
	if(1 == EDGEPOS(gPanelObj.KeyMatric[S$KEYMATRIX_SENSOR_UP ],PKeyMatric[S$KEYMATRIX_SENSOR_UP ]))
	{
		pMold->Sensor.Step = 15000;
	}

	if(1 == EDGENEG(gPanelObj.KeyMatric[S$KEYMATRIX_SENSOR_UP ],NKeyMatric[S$KEYMATRIX_SENSOR_UP ]))
	{
		pMold->Sensor.Step = 20000;
	}

	/*  ------------------------ sensor down -----------------------  */
	if(1 == EDGEPOS(gPanelObj.KeyMatric[S$KEYMATRIX_SENSOR_DN ],PKeyMatric[S$KEYMATRIX_SENSOR_DN ]))
	{
		pMold->Sensor.Step = 5000;
	}

	if(1 == EDGENEG(gPanelObj.KeyMatric[S$KEYMATRIX_SENSOR_DN ],NKeyMatric[S$KEYMATRIX_SENSOR_DN ]))
	{
		pMold->Sensor.Step = 20000;
	}

	/* ------------------------------ High blow air  ----------------------------- */
	if(1 == EDGEPOS(gPanelObj.KeyMatric[S$KEYMATRIX_BLOW],PKeyMatric[S$KEYMATRIX_BLOW]))
	{
		if (1 == gMachineOut.OilPump)
		{
			pMold->HighBlow.Step = 5000;
		}
		else
		{
			gImply.OilPumpNotOn  = !gMachineOut.OilPump;
		}
	}

	if(1 == EDGENEG(gPanelObj.KeyMatric[S$KEYMATRIX_BLOW],NKeyMatric[S$KEYMATRIX_BLOW]))
	{
		pMold->HighBlow.Step = 20000;
	}

	/* ------------------------------ Low blow air  ----------------------------- */
	if(1 == EDGEPOS(gPanelObj.KeyMatric[S$KEYMATRIX_BLOW_LOW   ],PKeyMatric[S$KEYMATRIX_BLOW_LOW   ]))
	{
		if(pMold->LowBlow.Step != 5000)
		{
			pMold->LowBlow.Step = 5000;
		}
		else
		{
			pMold->LowBlow.Step = 20000;
		}
	}

	/*if(1 == EDGENEG(gPanelObj.KeyMatric[S$KEYMATRIX_BLOW_LOW   ],NKeyMatric[S$KEYMATRIX_BLOW_LOW   ]))
	{
		pMold->LowBlow.Step = 20000;
	}*/

	/*  ------------------------   Extruder up -----------------------  */
	if(1 == EDGEPOS(gPanelObj.KeyMatric[S$KEYMATRIX_EXTRUDER_UP],PKeyMatric[S$KEYMATRIX_EXTRUDER_UP]))
	{
		if(pMold->Option.ExtrLift)
		{
			if (1 == gMachineOut.OilPump)
			{
				if( ACTUATOR_HYD  == gMachineFix.ExtrLift.eActuatorType )  // Hydraulic
				{
					if( 400 == pMold->ExtrLift.Step || 450 == pMold->ExtrLift.Step)// up -> stop
					{
						pMold->ExtrLift.Step = 0;/*Extruder stop*/
					}
					else
					{
						if((0 == pMold->TransDIn.ExtruderLiftUpLimit && 0 == pMold->TransDIn.ExtruderLiftDnLimit)
							|| 1 == pMold->TransDIn.ExtruderLiftUpLimit)
						{
							pMold->ExtrLift.Step = 10300;/*Extruder down*/
						}
						else
						{
							pMold->ExtrLift.Step = 300;/*Extruder up*/
						}
					}

				}
				else if(ACTUATOR_ELECTRIC  == gMachineFix.ExtrLift.eActuatorType)	//Electric
				{
					RMold.ExtrLift.Step = 5000;/*Extruder up*/
				}
			}
			else
			{
				gImply.OilPumpNotOn  = !gMachineOut.OilPump;
			}
		}
		else
		{
			gImply.NoFunction = 1;
		}

	}

	if( ACTUATOR_ELECTRIC  == gMachineFix.ExtrLift.eActuatorType )
	{
		if(1 == EDGENEG(gPanelObj.KeyMatric[S$KEYMATRIX_EXTRUDER_UP],NKeyMatric[S$KEYMATRIX_EXTRUDER_UP]))
		{
			RMold.ExtrLift.Step = 20000;
		}
	}
	/*  ------------------------   Extruder down (Electric) -----------------------  */
	if(1 == EDGEPOS(gPanelObj.KeyMatric[S$KEYMATRIX_EXTRUDER_DN],PKeyMatric[S$KEYMATRIX_EXTRUDER_DN]))
	{
		if(pMold->Option.ExtrLift)
		{
			if (1 == gMachineOut.OilPump)
			{
				if(ACTUATOR_ELECTRIC  == gMachineFix.ExtrLift.eActuatorType)
				{
					RMold.ExtrLift.Step = 15000;/*Extruder down*/
				}
			}
			else
			{
				gImply.OilPumpNotOn  = !gMachineOut.OilPump;
			}
		}
		else
		{
			gImply.NoFunction = 1;
		}
	}

	if( ACTUATOR_ELECTRIC  == gMachineFix.ExtrLift.eActuatorType )
	{
		if(1 == EDGENEG(gPanelObj.KeyMatric[S$KEYMATRIX_EXTRUDER_DN],NKeyMatric[S$KEYMATRIX_EXTRUDER_DN]))
		{
			RMold.ExtrLift.Step = 20000;
		}
	}

	/*------------------------Plate Up---------------------------------*/

	if(1 == EDGEPOS(gPanelObj.KeyMatric[S$KEYMATRIX_PLATE_UP  ],PKeyMatric[S$KEYMATRIX_PLATE_UP]))
	{

		if(1 == gMachineOut.OilPump)
		{
			if( 0 == gMachineIn.PlateUpLimit)
			{
				pMold->Plate.Step = 5000;
				gPanelObj.LedMatric[S$KEYMATRIX_PLATE_UP] = 1;
			}
			else
			{
				gImply.PlateUpLimit = gMachineIn.PlateUpLimit;
			}
		}
		else
		{
			gImply.OilPumpNotOn  = !gMachineOut.OilPump;
		}
	}
	if(1 == EDGENEG(gPanelObj.KeyMatric[S$KEYMATRIX_PLATE_UP  ],NKeyMatric[S$KEYMATRIX_PLATE_UP  ]))
	{
		pMold->Plate.Step = 20000;
		gPanelObj.LedMatric[S$KEYMATRIX_PLATE_UP] = 0;
	}

	/*------------------------Plate Down---------------------------------*/
	if(1 == EDGEPOS(gPanelObj.KeyMatric[S$KEYMATRIX_PLATE_DN  ],PKeyMatric[S$KEYMATRIX_PLATE_DN  ]))
	{
		if(1 == gMachineOut.OilPump)
		{
			if( 0 == gMachineIn.PlateDnLimit)
			{
				pMold->Plate.Step = 15000;
				gPanelObj.LedMatric[S$KEYMATRIX_PLATE_DN] = 1;
			}
			else
			{
				gImply.PlateDnLimit = gMachineIn.PlateDnLimit;
			}
		}
		else
		{
			gImply.OilPumpNotOn  = !gMachineOut.OilPump;
		}
	}
	if(1 == EDGENEG(gPanelObj.KeyMatric[S$KEYMATRIX_PLATE_DN  ],NKeyMatric[S$KEYMATRIX_PLATE_DN  ]))
	{
		pMold->Plate.Step = 20000;
		gPanelObj.LedMatric[S$KEYMATRIX_PLATE_DN] = 0;

	}

	/*------------------------Plate Fw---------------------------------*/

	if(1 == EDGEPOS(gPanelObj.KeyMatric[S$KEYMATRIX_PLATE_FW  ],PKeyMatric[S$KEYMATRIX_PLATE_FW]))
	{
		if(1 == gMachineOut.OilPump)
		{
			pMold->Plate.Step = 6100;
			gPanelObj.LedMatric[S$KEYMATRIX_PLATE_FW] = 1;
		}
		else
		{
			gImply.OilPumpNotOn  = !gMachineOut.OilPump;
		}
	}
	if(1 == EDGENEG(gPanelObj.KeyMatric[S$KEYMATRIX_PLATE_FW  ],NKeyMatric[S$KEYMATRIX_PLATE_FW  ]))
	{
		pMold->Plate.Step = 20000;
		gPanelObj.LedMatric[S$KEYMATRIX_PLATE_FW] = 0;
	}
	/*------------------------Plate Bw---------------------------------*/

	if(1 == EDGEPOS(gPanelObj.KeyMatric[S$KEYMATRIX_PLATE_BW  ],PKeyMatric[S$KEYMATRIX_PLATE_BW]))
	{
		if(1 == gMachineOut.OilPump)
		{
			pMold->Plate.Step = 16100;
			gPanelObj.LedMatric[S$KEYMATRIX_PLATE_BW] = 1;
		}
		else
		{
			gImply.OilPumpNotOn  = !gMachineOut.OilPump;
		}
	}
	if(1 == EDGENEG(gPanelObj.KeyMatric[S$KEYMATRIX_PLATE_BW  ],NKeyMatric[S$KEYMATRIX_PLATE_BW  ]))
	{
		pMold->Plate.Step = 20000;
		gPanelObj.LedMatric[S$KEYMATRIX_PLATE_BW] = 0;
	}

	/*------------------------------------------------------------------*/

	//	if(1 == EDGENEG(gPanelObj.KeyMatric[S$KEYMATRIX_EXTRUDER_UP],NKeyMatric[S$KEYMATRIX_EXTRUDER_UP]))
	//	{
	//		pMold->ExtrLift.Step = 20000;
	//	}
	/*  ------------------------   cutter -----------------------  */
	if(1 == EDGEPOS(gPanelObj.KeyMatric[S$KEYMATRIX_CUTTER_FW   ],PKeyMatric[S$KEYMATRIX_CUTTER_FW   ]))
	{
		//		gImply.DisableCutterCalibMode = 1;

		if (pMold->Option.Cutter)
		{
			if(1 == gMachineIn.SafeGate)
			{
				//			gThickIO.In.StartThick = 1;
				//			RMold.Cutter.Step = 100;
				////			gMachineOut.CutterFw = !gMachineOut.CutterFw;
				if (1 == gMachineOut.OilPump)
				{
					if(1 == gMachineFix.Option.bExtParisonCtrl)
					{
						gMachineInfo.ExtParisonCtrlStart = 1; /*   外部壁厚启动   */
					}
					else
					{
						gThickIO.In.StartThick = 1;      /*   壁厚启动   */
					}
					RMold.SupportAir.cntTime = gThickProf.TimSet.CycleTime;
					pMold->Cutter.Step = 300; //ipis20190131
					//	RMold.SupportAir.Step = 100;	 //ipis0304
				}
				else
				{
					gImply.OilPumpNotOn  = !gMachineOut.OilPump;
				}
			}
			else
			{
				gMachineOut.CutterFw = 0;
				gImply.SafeGate = 1;
			}
		}
		else
		{
			gImply.NoFunction = 1;
		}
	}

	/*  ------------------------   cool pin down -----------------------  */
	if(1 == EDGEPOS(gPanelObj.KeyMatric[S$KEYMATRIX_COOL_DN   ],PKeyMatric[S$KEYMATRIX_COOL_DN   ]))
	{
		if(pMold->Option.CoolPin)
		{
			if(1 == gMachineOut.OilPump)
			{
				if(1 == pMold->ValveOut.CoolPinDn) // Dn
				{
					pMold->CoolPin.Step = 15000;
				}
				else
				{
					pMold->CoolPin.Step = 5000;
				}
			}
			else
			{
				gImply.OilPumpNotOn  = !gMachineOut.OilPump;
			}
		}
		else
		{
			gImply.NoFunction = 1;
		}
	}

	/*  ------------------------   cool pin blow -----------------------  */
	if(1 == EDGEPOS(gPanelObj.KeyMatric[S$KEYMATRIX_COOL_BLOW   ],PKeyMatric[S$KEYMATRIX_COOL_BLOW   ]))
	{
		if(pMold->Option.CoolPin)
		{
			if(1 == gMachineOut.OilPump)
			{
				pMold->CoolPinBlow.Step = 5000;
			}
			else
			{
				gImply.OilPumpNotOn  = !gMachineOut.OilPump;
			}
		}
		else
		{
			gImply.NoFunction = 1;
			pMold->ValveOut.CoolPinBlow = 0;
		}
	}

	if(1 == EDGENEG(gPanelObj.KeyMatric[S$KEYMATRIX_COOL_BLOW  ],NKeyMatric[S$KEYMATRIX_COOL_BLOW  ]))
	{
		pMold->CoolPinBlow.Step = 20000;
	}

	/*  ------------------------   cool pin 2 down -----------------------  */
	if(1 == EDGEPOS(gPanelObj.KeyMatric[S$KEYMATRIX_COOL2_DN   ],PKeyMatric[S$KEYMATRIX_COOL2_DN   ]))
	{
		if(pMold->Option.CoolPin2)
		{
			if(1 == gMachineOut.OilPump)
			{
				if(1 == pMold->ValveOut.CoolPin2Dn) // Dn
				{
					pMold->CoolPin2.Step = 15000;
				}
				else
				{
					pMold->CoolPin2.Step = 5000;
				}
			}
			else
			{
				gImply.OilPumpNotOn  = !gMachineOut.OilPump;
			}
		}
		else
		{
			gImply.NoFunction = 1;
		}
	}
	/*  ------------------------   cool pin 2 Blow -----------------------  */
	if(1 == EDGEPOS(gPanelObj.KeyMatric[S$KEYMATRIX_COOL2_BLOW   ],PKeyMatric[S$KEYMATRIX_COOL2_BLOW   ]))
	{
		if(pMold->Option.CoolPin2)
		{
			if(1 == gMachineOut.OilPump)
			{
				pMold->CoolPin2Blow.Step = 5000;
			}
			else
			{
				gImply.OilPumpNotOn  = !gMachineOut.OilPump;
			}
		}
		else
		{
			gImply.NoFunction = 1;
			pMold->ValveOut.CoolPin2Blow = 0;
		}

	}

	if(1 == EDGENEG(gPanelObj.KeyMatric[S$KEYMATRIX_COOL2_BLOW  ],NKeyMatric[S$KEYMATRIX_COOL2_BLOW  ]))
	{
		pMold->CoolPin2Blow.Step = 20000;
	}

	/*  ------------------------   cool pin 3 down -----------------------  */
	if(1 == EDGEPOS(gPanelObj.KeyMatric[S$KEYMATRIX_COOL3_DN   ],PKeyMatric[S$KEYMATRIX_COOL3_DN   ]))
	{
		if(pMold->Option.CoolPin3)
		{
			if(1 == gMachineOut.OilPump)
			{
				if(1 == pMold->ValveOut.CoolPin3Dn) // Dn
				{
					pMold->CoolPin3.Step = 15000;
				}
				else
				{
					pMold->CoolPin3.Step = 5000;
				}
			}
			else
			{
				gImply.OilPumpNotOn  = !gMachineOut.OilPump;
			}
		}
		else
		{
			gImply.NoFunction = 1;
		}
	}

	/*  ------------------------   cool pin 3 Blow -----------------------  */
	if(1 == EDGEPOS(gPanelObj.KeyMatric[S$KEYMATRIX_COOL3_BLOW   ],PKeyMatric[S$KEYMATRIX_COOL3_BLOW   ]))
	{
		if(pMold->Option.CoolPin3)
		{
			if(1 == gMachineOut.OilPump)
			{
				pMold->CoolPin3Blow.Step = 5000;
			}
			else
			{
				gImply.OilPumpNotOn  = !gMachineOut.OilPump;
			}
		}
		else
		{
			gImply.NoFunction = 1;
			pMold->ValveOut.CoolPin3Blow = 0;
		}
	}

	if(1 == EDGENEG(gPanelObj.KeyMatric[S$KEYMATRIX_COOL3_BLOW  ],NKeyMatric[S$KEYMATRIX_COOL3_BLOW  ]))
	{
		pMold->CoolPin3Blow.Step = 20000;
	}

	/*------------------------Blow Pin Down Hold ---------------------------------*/
	if(1 == EDGEPOS(gPanelObj.KeyMatric[S$KEYMATRIX_BLOWPINDN_HOLD  ],PKeyMatric[S$KEYMATRIX_BLOWPINDN_HOLD  ]))
	{
		if(1 == gMachineOut.OilPump)
		{
			if (1==pMold->BlowPin.UpPos)
			{
				//	pMold->BlowPin.Step = 19000;
				pMold->ValveOut.BlowPinDnHold = !pMold->ValveOut.BlowPinDnHold;
			}
			else
			{
				if(pMold == & LMold)
				{
					gImply.LPinUp      = !pMold->BlowPin.UpPos;
				}
				else
				{
					gImply.RPinUp      = !pMold->BlowPin.UpPos;
				}
			}
		}
		else
		{
			gImply.OilPumpNotOn  = !gMachineOut.OilPump;
			gHardWare.XP0101Led_1[2] =1;
		}

	}
	//	if(1 == EDGENEG(gPanelObj.KeyMatric[S$KEYMATRIX_BLOWPINDN_HOLD  ],NKeyMatric[S$KEYMATRIX_BLOWPINDN_HOLD  ]))
	//		{
	//		pMold->BlowPin.Step = 20000;
	//		gHardWare.XP0101Led_1[2] =0;
	//	}

	/*  ------------------------   Hook pin Fw -----------------------  */
	if(1 == EDGEPOS(gPanelObj.KeyMatric[S$KEYMATRIX_HOOK_PIN_FW   ],PKeyMatric[S$KEYMATRIX_HOOK_PIN_FW   ]))
	{
		if(pMold->Option.HookPin)
		{
			if(1 == gMachineOut.OilPump)
			{
				if(1 == pMold->ValveOut.HookPinFw) // Fw
				{
					pMold->HookPin.Step = 15000;
				}
				else
				{
					if(1 == pMold->TransDIn.CarriageBwLimit)
					{
						pMold->HookPin.Step = 5000;
					}
					else
					{
						if(pMold == & LMold)
						{
							gImply.LCarriageBw = !pMold->TransDIn.CarriageBwLimit;
						}
						else
						{
							gImply.RCarriageBw = !pMold->TransDIn.CarriageBwLimit;
						}
					}
				}
			}
			else
			{
				gImply.OilPumpNotOn  = !gMachineOut.OilPump;
			}
		}
		else
		{
			gImply.NoFunction = 1;
		}
	}

	/* ------------------------------  Deflasher handle ----------------------------- */
	if(1 == EDGEPOS(gPanelObj.KeyMatric[S$KEYMATRIX_HANDLE_PUNCHER   ],PKeyMatric[S$KEYMATRIX_HANDLE_PUNCHER   ]))
	{
		if(pMold->Option.PunchHandle)
		{
			if(1 == gMachineOut.OilPump)
			{

				if (1 == pMold->TransDIn.TopDeflashFwLimit)
				{
					pMold->ValveOut.TopDeflashCls = !pMold->ValveOut.TopDeflashCls;
				}
				else
				{
					if(pMold == & LMold)
					{
						gImply.LTopDeflashFw = 1;
					}
					else
					{
						gImply.RTopDeflashFw = 1;
					}
				}
			}
			else
			{
				gImply.OilPumpNotOn  = !gMachineOut.OilPump;
			}
		}
		else
		{
			gImply.NoFunction = 1;
			pMold->ValveOut.TopDeflashCls = 0;
		}
	}

	//	if(1 == EDGENEG(gPanelObj.KeyMatric[S$KEYMATRIX_CUTTER_FW],NKeyMatric[S$KEYMATRIX_CUTTER_FW]))
	//	{
	//		RMold.Cutter.Step = 20000;
	//	}
}/* end of CalibCtrl( Mold_typ *pMold)  */
/* ------------------------------------------------------------------*/

void CalibRLCtrl( Mold_typ *pMold)
{
	/*  ------------------------   cutter -----------------------  */
	if(1 == EDGEPOS(gPanelObj.KeyMatric[S$KEYMATRIX_CUTTER_FW   ],PKeyMatric[S$KEYMATRIX_CUTTER_FW   ]))
	{
		if (pMold->Option.Cutter)
		{
			if(1 == gMachineIn.SafeGate)
			{
				//			gThickIO.In.StartThick = 1;
				//			RMold.Cutter.Step = 100;
				////			gMachineOut.CutterFw = !gMachineOut.CutterFw;
				if (1 == gMachineOut.OilPump)
				{
					if(1 == gMachineFix.Option.bExtParisonCtrl)
					{
						gMachineInfo.ExtParisonCtrlStart = 1; /*   外部壁厚启动   */
					}
					else
					{
						gThickIO.In.StartThick = 1;      /*   壁厚启动   */
					}
					RMold.SupportAir.cntTime = gThickProf.TimSet.CycleTime;
					RMold.Cutter.Step = 300; //ipis20190131
					//	RMold.SupportAir.Step = 100;	 //ipis0304
				}
				else
				{
					gImply.OilPumpNotOn  = !gMachineOut.OilPump;
				}
			}
			else
			{
				gMachineOut.CutterFw = 0;
				gImply.SafeGate = 1;
			}
		}
		else
		{
			gImply.NoFunction = 1;
		}
	}

	/*  ------------------------   Extruder up -----------------------  */
	if(1 == EDGEPOS(gPanelObj.KeyMatric[S$KEYMATRIX_EXTRUDER_UP],PKeyMatric[S$KEYMATRIX_EXTRUDER_UP]))
		{
		if(pMold->Option.ExtrLift)
		{
			if (1 == gMachineOut.OilPump)
			{
				if( ACTUATOR_HYD  == gMachineFix.ExtrLift.eActuatorType )  // Hydraulic
				{
					if((0 == pMold->TransDIn.ExtruderLiftUpLimit && 0 == pMold->TransDIn.ExtruderLiftDnLimit)
						|| 1 == pMold->TransDIn.ExtruderLiftUpLimit)
					{
						pMold->ExtrLift.Step = 10300;/*Extruder down*/
					}
					else
					{
						pMold->ExtrLift.Step = 300;/*Extruder up*/
					}
				}
				else if(ACTUATOR_ELECTRIC  == gMachineFix.ExtrLift.eActuatorType)	//Electric
				{
					RMold.ExtrLift.Step = 5000;/*Extruder up*/
				}
			}
			else
			{
				gImply.OilPumpNotOn  = !gMachineOut.OilPump;
			}
		}
		else
		{
			gImply.NoFunction = 1;
		}

	}

	if( ACTUATOR_ELECTRIC  == gMachineFix.ExtrLift.eActuatorType )
	{
		if(1 == EDGENEG(gPanelObj.KeyMatric[S$KEYMATRIX_EXTRUDER_UP],NKeyMatric[S$KEYMATRIX_EXTRUDER_UP]))
			{
			RMold.ExtrLift.Step = 20000;
		}
	}
	/*  ------------------------   Extruder down (Electric) -----------------------  */
	if(1 == EDGEPOS(gPanelObj.KeyMatric[S$KEYMATRIX_EXTRUDER_DN],PKeyMatric[S$KEYMATRIX_EXTRUDER_DN]))
		{
		if(pMold->Option.ExtrLift)
		{
			if (1 == gMachineOut.OilPump)
			{
				if(ACTUATOR_ELECTRIC  == gMachineFix.ExtrLift.eActuatorType)
				{
					RMold.ExtrLift.Step = 15000;/*Extruder down*/
				}
			}
			else
			{
				gImply.OilPumpNotOn  = !gMachineOut.OilPump;
			}
		}
		else
		{
			gImply.NoFunction = 1;
		}
	}

	if( ACTUATOR_ELECTRIC  == gMachineFix.ExtrLift.eActuatorType )
	{
		if(1 == EDGENEG(gPanelObj.KeyMatric[S$KEYMATRIX_EXTRUDER_DN],NKeyMatric[S$KEYMATRIX_EXTRUDER_DN]))
		{
			RMold.ExtrLift.Step = 20000;
		}
	}

	/*------------------------Plate Up---------------------------------*/

	if(1 == EDGEPOS(gPanelObj.KeyMatric[S$KEYMATRIX_PLATE_UP  ],PKeyMatric[S$KEYMATRIX_PLATE_UP]))
	{
		if(1 == gMachineOut.OilPump)
		{
			if( 0 == gMachineIn.PlateUpLimit)
			{
				pMold->Plate.Step = 5000;
				gPanelObj.LedMatric[S$KEYMATRIX_PLATE_UP] = 1;
			}
			else
			{
				gImply.PlateUpLimit = gMachineIn.PlateUpLimit;
			}
		}
		else
		{
			gImply.OilPumpNotOn  = !gMachineOut.OilPump;
		}
	}
	if(1 == EDGENEG(gPanelObj.KeyMatric[S$KEYMATRIX_PLATE_UP  ],NKeyMatric[S$KEYMATRIX_PLATE_UP  ]))
	{
		pMold->Plate.Step = 20000;
		gPanelObj.LedMatric[S$KEYMATRIX_PLATE_UP] = 0;
	}

	/*------------------------Plate Down---------------------------------*/
	if(1 == EDGEPOS(gPanelObj.KeyMatric[S$KEYMATRIX_PLATE_DN  ],PKeyMatric[S$KEYMATRIX_PLATE_DN  ]))
	{
		if(1 == gMachineOut.OilPump)
		{
			if( 0 == gMachineIn.PlateDnLimit)
			{
				pMold->Plate.Step = 15000;
				gPanelObj.LedMatric[S$KEYMATRIX_PLATE_DN] = 1;
			}
			else
			{
				gImply.PlateDnLimit = gMachineIn.PlateDnLimit;
			}
		}
		else
		{
			gImply.OilPumpNotOn  = !gMachineOut.OilPump;
		}
	}
	if(1 == EDGENEG(gPanelObj.KeyMatric[S$KEYMATRIX_PLATE_DN  ],NKeyMatric[S$KEYMATRIX_PLATE_DN  ]))
	{
		pMold->Plate.Step = 20000;
		gPanelObj.LedMatric[S$KEYMATRIX_PLATE_DN] = 0;

	}

	/*------------------------Plate Fw---------------------------------*/

	if(1 == EDGEPOS(gPanelObj.KeyMatric[S$KEYMATRIX_PLATE_FW  ],PKeyMatric[S$KEYMATRIX_PLATE_FW]))
	{
		if(1 == gMachineOut.OilPump)
		{
			pMold->Plate.Step = 6100;
			gPanelObj.LedMatric[S$KEYMATRIX_PLATE_FW] = 1;
		}
		else
		{
			gImply.OilPumpNotOn  = !gMachineOut.OilPump;
		}
	}
	if(1 == EDGENEG(gPanelObj.KeyMatric[S$KEYMATRIX_PLATE_FW  ],NKeyMatric[S$KEYMATRIX_PLATE_FW  ]))
	{
		pMold->Plate.Step = 20000;
		gPanelObj.LedMatric[S$KEYMATRIX_PLATE_FW] = 0;
	}
	/*------------------------Plate Bw---------------------------------*/

	if(1 == EDGEPOS(gPanelObj.KeyMatric[S$KEYMATRIX_PLATE_BW  ],PKeyMatric[S$KEYMATRIX_PLATE_BW]))
	{
		if(1 == gMachineOut.OilPump)
		{
			pMold->Plate.Step = 16100;
			gPanelObj.LedMatric[S$KEYMATRIX_PLATE_BW] = 1;
		}
		else
		{
			gImply.OilPumpNotOn  = !gMachineOut.OilPump;
		}
	}
	if(1 == EDGENEG(gPanelObj.KeyMatric[S$KEYMATRIX_PLATE_BW  ],NKeyMatric[S$KEYMATRIX_PLATE_BW  ]))
	{
		pMold->Plate.Step = 20000;
		gPanelObj.LedMatric[S$KEYMATRIX_PLATE_BW] = 0;
	}

}/* end of ManualCtrl( Mold_typ *pMold)  */
```

#### calib.var
```iecst
VAR
	t_init : USINT;
	t_stop : USINT;
	Init : USINT;
	PKeyMatric : ARRAY[0..MAX_KEY_COUNT] OF USINT;
	NKeyMatric : ARRAY[0..MAX_KEY_COUNT] OF USINT;
	MachineInOld : Machine_In_typ;
	MachineInOldN : Machine_In_typ;
	OldRClampOpnDI : USINT;
	OldLClampOpnDI : USINT;
END_VAR
```

- defines.h (reference to Logical/GlobalIncludes/defines.h)

- edge.h (reference to Logical/GlobalIncludes/edge.h)

- pic_id.h (reference to Logical/GlobalIncludes/pic_id.h)

- keyap880.h (reference to Logical/GlobalIncludes/keyap880.h)

### Program Logical/machine/reset (ANSIC, version 1.00.0) - machine reset task

#### reset.c
```c
/********************************************************************
 * COPYRIGHT --  B&R China
 ********************************************************************
 * Program: reset
 * File: reset.c
 * Author: lijianjun
 * Created: March 06, 2013
 ********************************************************************
 * Implementation of program reset --- machine reset control
 ********************************************************************/

#include <bur/plctypes.h>

#ifdef _DEFAULT_INCLUDES
#include <AsDefault.h>
#endif

/**************************************************************************************
                            Function Declarations
**************************************************************************************/

void MoldReset( Mold_typ * pMold);
void MoldReset_Hybrid(Mold_typ * pMold);

/**************************************************************************************
     	        		I N I T U P  O F   T H E   T A S K
**************************************************************************************/
_INIT void init ( void )
{
	LMold.ResetStep = 0;
	RMold.ResetStep = 0;
} /* end of _INIT */

 /*************************************************************************************
        				C Y C L I C   P A R T   O F   T H E   T A S K
**************************************************************************************/

_CYCLIC void cyclic ( void )
{
	if(LMold.TimeSet.ResetAlarmTime < 1)LMold.TimeSet.ResetAlarmTime = 2000;
	if(RMold.TimeSet.ResetAlarmTime < 1)RMold.TimeSet.ResetAlarmTime = 2000;

	MoldReset_Hybrid(&RMold);
	MoldReset_Hybrid(&LMold);

} /* end of _CYCLIC */

void MoldReset_Hybrid( Mold_typ * pMold)
{
	if(0 == gMachineIn.SafeGate)
	{
		if(pMold->ResetStep > 100 && pMold->ResetStep < 3000 )
		{
			pMold->ResetStep = 20000;
		}
	}

	switch (pMold->ResetStep)
	{
		case 100:/*Blow Pin Up, extruderlift down*/
			pMold->TimeCycle.IN   = 1;
			pMold->TimeCycle.PT   = pMold->TimeSet.ResetAlarmTime;	/*  限时  */
			pMold->ValveOut.ProductAuxClamp =0;

			if(ACTUATOR_ELECTRIC == gMachineFix.ExtrLift.eActuatorType)
			{
				RMold.ExtrLift.Step = 10300;/*Exturderlif down*/
			}
			else
			{
				pMold->ExtrLift.Step = 10300;/*Exturderlif down*/
			}

			if(pMold->Carriage.BwPos
				&& pMold->Clamp.OpnPos
				&& pMold->TransDIn.CoolPinUpLimit && pMold->TransDIn.CoolPin2UpLimit && pMold->TransDIn.CoolPin3UpLimit
				&& pMold->TransDIn.TopDeflashBwLimit && pMold->TransDIn.BottomDeflashBwLimit
				&& pMold->TransDIn.TopDeflashOpnLimit
				&& pMold->TransDIn.RobotBwLimit && pMold->TransDIn.RobotUpLimit
				&& pMold->TransDIn.RobotOpnLimit
				&& pMold->TransDIn.SubMoldClsLimit && pMold->TransDIn.BottomSubMoldClsLimit
				&& pMold->TransDIn.HookPinBwLimit
				//		&& pMold->TransDIn.PinPartFwLimit
				//	    && pMold->TransDIn.RobotOpnLimit
				//	    && pMold->TransDIn.CutNeckOpnLimit
				//		&& pMold->TransDIn.SealOpnLimit
				&& pMold->Robot.Transfer.BwPos
				&& (pMold->Robot.Transfer.CalOK || ACTUATOR_ELECTRIC != gMachineFix.MoldR.RobotTransfer.eValveType)
				&& pMold->Robot.UpDn.UpPos
				&& (pMold->Robot.UpDn.CalOK || ACTUATOR_ELECTRIC != gMachineFix.MoldR.RobotUpDn.eValveType)
				&& pMold->TransDIn.RobotOpnLimit
				//		&& pMold->TransDIn.RobotOpnLimitL
				//		&& pMold->TransDIn.RobotOpnLimitR
				)
			{
				pMold->ResetStep = 1290;  /* jump reset process*/
			}
			else if(0 == pMold->BlowPin.UpPos || 0 == pMold->BlowPin2.UpPos)
			{
				pMold->BlowPin.Step = 10300;    /*  吹针上    */
				pMold->BlowPin2.Step = 10300;    /*  吹针上    */

				pMold->ResetStep = 200;
			}
			else
			{
				pMold->ResetStep = 210;
			}
			break;

		case 200:/*wait blow pin up finished*/
			if( 13000 == pMold->BlowPin.Step && 13000 == pMold->BlowPin2.Step )	/*  吹针上   */
			{
				pMold->BlowPin.Step = 0;
				pMold->BlowPin2.Step = 0;
				pMold->ResetStep = 210;
			}

			if(40000 == pMold->BlowPin.Step)
			{
				pMold->BlowPin.Step = 0;
				pMold->ResetStep = 40000;
			}

			if(40000 == pMold->BlowPin2.Step)
			{
				pMold->BlowPin2.Step = 0;
				pMold->ResetStep = 40000;
			}

			break;

		case 210:

			if(ACTUATOR_ELECTRIC == gMachineFix.ExtrLift.eActuatorType)
			{
				if (13000==pMold->ExtrLift.Step)
				{
					RMold.ExtrLift.Step =0;
					pMold->ResetStep = 250;
				}

				if (40000==pMold->ExtrLift.Step)
				{
					RMold.ExtrLift.Step =0;
					pMold->ResetStep = 40000;
				}
			}
			else
			{
				if (13000==pMold->ExtrLift.Step)
				{
					pMold->ExtrLift.Step =0;
					pMold->ResetStep = 250;
				}

				if (40000==pMold->ExtrLift.Step)
				{
					pMold->ExtrLift.Step =0;
					pMold->ResetStep = 40000;
				}
			}
			break;

		case 250:/*TopDeflash open (handle backward)  打手挽退+打手把退*/
			pMold->ValveOut.BlowPinDnHold =0;
			if((1 == pMold->Option.PunchHandle) && (0 == pMold->TransDIn.TopDeflashOpnLimit))
				//	if((0 == pMold->TransDIn.TopDeflashOpnLimit))
			{
				pMold->TopDeflash.Step = 1100;
				pMold->ResetStep = 260;
			}
			else
			{
				pMold->ResetStep = 300;
			}

			break;

		case 260:

			if(3000 == pMold->TopDeflash.Step)
			{
				pMold->TopDeflash.Step = 0;
				pMold->ResetStep = 300;
			}

			if(40000 == pMold->TopDeflash.Step)
			{
				pMold->TopDeflash.Step = 0;
				pMold->ResetStep = 40000;
			}

			break;

		case 300:/*TopDeflash Backward*/
			//	if((1 == pMold->Option.TopDeflash) && (0 == pMold->TransDIn.TopDeflashBwLimit))
			if(0 == pMold->TransDIn.TopDeflashBwLimit)
			{
				pMold->TopDeflash.Step = 1300;
				pMold->ResetStep = 310;
			}
			else
			{
				pMold->ResetStep = 400;
			}
			break;

		case 310:/*wait topdeflash backward finish*/
			if(3000 == pMold->TopDeflash.Step)
			{
				pMold->TopDeflash.Step = 0;
				pMold->ResetStep = 400;
			}

			if(40000 == pMold->TopDeflash.Step)
			{
				pMold->TopDeflash.Step = 0;
				pMold->ResetStep = 40000;
			}
			break;

		case 400:/*BottomDeflash Backward*/
			//	if((1 == pMold->Option.BottomDeflash) && (0 == pMold->TransDIn.BottomDeflashBwLimit))
			if(0 == pMold->TransDIn.BottomDeflashBwLimit)
			{
				pMold->BottomDeflash.Step = 1300;
				pMold->ResetStep = 410;
			}
			else
			{
				pMold->ResetStep = 500;
			}
			break;

		case 410:/*wait BottomDeflash backward finish*/
			if(3000 == pMold->BottomDeflash.Step)
			{
				pMold->BottomDeflash.Step = 0;
				pMold->ResetStep = 500;
			}

			if(40000 == pMold->BottomDeflash.Step)
			{
				pMold->BottomDeflash.Step = 0;
				pMold->ResetStep = 40000;
			}
			break;

		case 500:/*CoolPin UP*/
			pMold->CoolPin.Step = 500;
			pMold->CoolPin2.Step = 500;
			pMold->CoolPin3.Step = 500;

			pMold->ResetStep = 510;
			break;

		case 510:/*wait CoolPin UP finish*/
			if(3000 == pMold->CoolPin.Step && 3000 == pMold->CoolPin2.Step && 3000 == pMold->CoolPin3.Step )
			{
				pMold->CoolPin.Step = 0;
				pMold->CoolPin2.Step = 0;
				pMold->CoolPin3.Step = 0;
				pMold->ResetStep = 600;
			}

			if(40000 == pMold->CoolPin.Step || 40000 == pMold->CoolPin2.Step || 40000 == pMold->CoolPin3.Step)
			{
				pMold->CoolPin.Step = 0;
				pMold->CoolPin2.Step = 0;
				pMold->CoolPin3.Step = 0;
				pMold->ResetStep = 40000;
			}

			break;

		case 600:/*HookPin Backward*/
			if(0 == pMold->TransDIn.HookPinBwLimit)
			{
				pMold->HookPin.Step = 1300;
				pMold->ResetStep = 610;
			}
			else
			{
				pMold->ResetStep = 700;
			}
			break;

		case 610:/*wait HookPin backward finish*/
			if(3000 == pMold->HookPin.Step)
			{
				pMold->BottomDeflash.Step = 0;
				pMold->ResetStep = 700;
			}

			if(40000 == pMold->HookPin.Step)
			{
				pMold->HookPin.Step = 0;
				pMold->ResetStep = 40000;
			}
			break;

		case 700:/*Clamp UnLock*/
			if(0 == pMold->Clamp.OpnPos)
			{
				pMold->Clamp.Step = 12100;		/*UnLock Process  開模洩壓 */
				pMold->ResetStep  = 710;
			}
			else
			{

				pMold->ResetStep  = 800;
			}
			break;

		case 710:/*wait UnLock finish*/
			if(13000 == pMold->Clamp.Step)
			{
				pMold->Clamp.Step = 0;
				pMold->ResetStep  = 750;
			}

			if(40000 == pMold->Clamp.Step)
			{
				pMold->Clamp.Step = 0;
				pMold->ResetStep  = 40000;
			}
			break;

		case 750:/*Clamp Open*/
			if(0 == pMold->Clamp.OpnPos)
			{
				pMold->Clamp.Step = 10300;		/*Clamp Open*/
				pMold->ResetStep  = 760;
			}
			else
			{
				pMold->ResetStep  = 900;
			}
			break;

		case 760:/*wait clamp open finish*/
			if(13000 == pMold->Clamp.Step)
			{
				pMold->Clamp.Step = 0;
				pMold->ResetStep  = 800;
			}

			if(40000 == pMold->Clamp.Step)
			{
				pMold->Clamp.Step = 0;
				pMold->ResetStep  = 40000;
			}
			break;

		case 800:  // Submold cls

			pMold->SubMold.Step  = 300;
			pMold->BottomSubMold.Step  = 300;
			pMold->ResetStep  = 810;

			break;

		case 810:
			if(3000 == pMold->SubMold.Step && 3000 == pMold->BottomSubMold.Step )
			{
				pMold->SubMold.Step = 0;
				pMold->BottomSubMold.Step =0;
				pMold->ResetStep  = 900;
			}

			if(40000 == pMold->SubMold.Step || 40000==pMold->BottomSubMold.Step)
			{
				pMold->SubMold.Step = 0;
				pMold->BottomSubMold.Step =0;
				pMold->ResetStep  = 40000;
			}
			break;

		case 900: // robot bw
			if(0 == pMold->Robot.Transfer.BwPos)
			{
				pMold->Robot.Step = 10300;
				pMold->ResetStep = 910;
			}
			else
			{
				pMold->ResetStep = 1000;
			}
			break;

		case 910:
			if(13000 == pMold->Robot.Step)
			{
				pMold->Robot.Step = 0;
				pMold->ResetStep  = 1000;
			}

			if(40000 == pMold->Robot.Step)
			{
				pMold->Robot.Step = 0;
				pMold->ResetStep  = 40000;
			}
			break;

		case 1000: // robot opn
			if(0 == pMold->TransDIn.RobotOpnLimit)
			{
				pMold->RobotOpnCls.Step = 10300;
				pMold->ResetStep = 1010;
			}
			else
			{
				pMold->ResetStep = 1100;
			}
			break;

		case 1010:
			if(13000 == pMold->RobotOpnCls.Step)
			{
				pMold->RobotOpnCls.Step = 0;
				pMold->ResetStep  = 1100;
			}

			if(40000 == pMold->RobotOpnCls.Step)
			{
				pMold->RobotOpnCls.Step = 0;
				pMold->ResetStep  = 40000;
			}
			break;

		case 1100:/*Carriage down backward*/
			if(0 == pMold->Carriage.BwPos)
			{
				pMold->Carriage.Step = 10300;
				pMold->ResetStep = 1110;
			}
			else
			{
				pMold->ResetStep = 1300;
			}
			break;

		case 1110:/*wait carriage down finish*/
			if(13000 == pMold->Carriage.Step)
			{
				pMold->Carriage.Step = 0;
				pMold->ResetStep = 1300;
			}

			if(40000 == pMold->Carriage.Step)
			{
				pMold->Carriage.Step = 0;
				pMold->ResetStep = 40000;
			}
			break;

		case 1290: // jump reset process

			if(ACTUATOR_ELECTRIC == gMachineFix.ExtrLift.eActuatorType)
			{
				if (13000==pMold->ExtrLift.Step)
				{
					RMold.ExtrLift.Step =0;
					pMold->ResetStep = 1300;
				}

				if (40000==pMold->ExtrLift.Step)
				{
					RMold.ExtrLift.Step =0;
					pMold->ResetStep = 40000;
				}
			}
			else
			{
				if (13000==pMold->ExtrLift.Step)
				{
					pMold->ExtrLift.Step =0;
					pMold->ResetStep = 1300;
				}

				if (40000==pMold->ExtrLift.Step)
				{
					pMold->ExtrLift.Step =0;
					pMold->ResetStep = 40000;
				}
			}

			break;

		case 1300:/*blowpin down*/

			if(0 == pMold->BlowPin.DnPos || 0 == pMold->BlowPin2.DnPos)
			{
				pMold->BlowPin.Step = 300;
				pMold->BlowPin2.Step = 300;
				pMold->ResetStep = 1310;
			}
			else
			{
				pMold->ResetStep = 1400;
			}

			break;

		case 1310:/*wait blowpin down finish*/

			if(3000 == pMold->BlowPin.Step && 3000 == pMold->BlowPin2.Step)
			{
				pMold->BlowPin.Step = 0;
				pMold->BlowPin2.Step = 0;
				pMold->ResetStep = 1400;
			}

			if(40000 == pMold->BlowPin.Step)
			{
				pMold->BlowPin.Step = 0;
				pMold->ResetStep = 40000;
			}

			if(40000 == pMold->BlowPin2.Step)
			{
				pMold->BlowPin2.Step = 0;
				pMold->ResetStep = 40000;
			}
			break;

		case 1400:

			pMold->TimeCycle.IN = 0;
			pMold->ResetStep = 3000;
			break;

		case 3000:
			break;

		case 20000:
			pMold->TimeCycle.IN = 0;

			pMold->LowBlow.Step			= 30000;
			pMold->HighBlow.Step			= 30000;
			pMold->BlowPin.Step			= 30000;
			pMold->BlowPin2.Step			= 30000;
			pMold->BottomPin.Step		= 30000;
			pMold->Carriage.Step		   = 20000;
			pMold->Clamp.Step			   = 30000;
			//	pMold->CoolPin.Step			= 30000;
			pMold->CoolPinBlow.Step	   = 30000;
			//	pMold->CoolPin2.Step		   = 30000;
			pMold->CoolPin2Blow.Step	= 30000;
			//	pMold->CoolPin3.Step	      = 30000;
			pMold->CoolPin3Blow.Step	= 30000;
			pMold->BlowDeflash.Step		= 30000;
			pMold->CoolDeflash.Step		= 30000;
			pMold->Cutter.Step			= 30000;
			pMold->TopDeflash.Step		= 30000;
			pMold->BottomDeflash.Step	= 30000;
			pMold->SupportAir.Step		= 30000;
			pMold->SupportSuckAir.Step		= 30000;
			if(ACTUATOR_ELECTRIC == gMachineFix.ExtrLift.eActuatorType) RMold.ExtrLift.Step		   = 30000;
			else  pMold->ExtrLift.Step		   = 30000;
			pMold->Lock.Step			   = 30000;
			pMold->PullBottom.Step		= 30000;
			pMold->InnerPin.Step	      = 30000;
			pMold->CutNeck.Step   		= 30000;
			//	pMold->Robot.Step	    	   = 30000;
			pMold->ChuteDeflashBlow.Step = 30000;
			pMold->SubMold.Step		   = 30000;
			pMold->PinPart.Step		   = 30000;
			pMold->Screw.Step		      = 30000;
			pMold->HookPin.Step		   = 30000;

			pMold->ResetStep = 0;
			break;

		case 30000:
			pMold->TimeCycle.IN = 0;
			pMold->ResetStep = 0;
			break;

		case 40000:
			pMold->TimeCycle.IN = 0;

			pMold->LowBlow.Step			= 30000;
			pMold->HighBlow.Step		= 30000;
			pMold->BlowPin.Step			= 30000;
			pMold->BlowPin2.Step		= 30000;
			pMold->BottomPin.Step		= 30000;
			pMold->Carriage.Step		= 20000;
			pMold->Clamp.Step			= 30000;
			pMold->CoolPin.Step			= 30000;
			pMold->CoolPinBlow.Step	    = 30000;
			pMold->CoolPin2.Step		= 30000;
			pMold->CoolPin2Blow.Step	= 30000;
			pMold->CoolPin3.Step	    = 30000;
			pMold->CoolPin3Blow.Step	= 30000;
			pMold->BlowDeflash.Step		= 30000;
			pMold->CoolDeflash.Step		= 30000;
			pMold->Cutter.Step			= 30000;
			pMold->TopDeflash.Step		= 30000;
			pMold->BottomDeflash.Step	= 30000;
			pMold->SupportAir.Step		= 30000;
			pMold->SupportSuckAir.Step	= 30000;
			if(ACTUATOR_ELECTRIC == gMachineFix.ExtrLift.eActuatorType) RMold.ExtrLift.Step		   = 30000;
			else  pMold->ExtrLift.Step	= 30000;
			pMold->Lock.Step			= 30000;
			pMold->PullBottom.Step		= 30000;
			pMold->InnerPin.Step	    = 30000;
			pMold->CutNeck.Step   		= 30000;
			pMold->Robot.Step	    	= 30000;
			pMold->ChuteDeflashBlow.Step = 30000;
			pMold->SubMold.Step		    = 30000;
			pMold->PinPart.Step		    = 30000;
			pMold->Screw.Step		    = 30000;
			pMold->HookPin.Step		    = 30000;

			pMold->ResetStep = 60000;
			break;

		case 60000:
			break;
	}/* end of switch */

	if(1 == gMachineInfo.MachineReset)
	{
		pMold->TimeDis.ResetAlarmTime = pMold->TimeCycle.ET;
	}

	//	if(1 == gMachineInfo.Manual && 1 == pMold->TimeCycle.IN)
	//	{
	//		pMold->TimeDis.CycleAlarmTime = pMold->TimeCycle.ET;
	//	}

	/* 单模复位限时到  */
	if(1 == pMold->TimeCycle.Q)
	{
		pMold->TimeCycle.IN = 0;
		pMold->ResetStep = 40000;
	}
}/*end of function */
```

### Program Logical/machine/manual (ANSIC, version 1.00.0) - manual task
